// TIA Portal project "磬苑一队（6部十层）" (V15.1)

(* hardware
DEVICE "S7-1200 station_1"  S7-1200 Station
   slot 0: "Rack_0"  S7-1200 Rack  Rack  V1.0
   slot 1: "PLC_1"  CPU 1215C DC/DC/DC  6ES7 215-1AG40-0XB0  V4.2
DEVICE "PC-System_1"  SIMATIC PC station
   slot 0: "SIMATIC PC station"  Rail  SIMATIC PC-Station  V1.0
      slot 125: "Stationmanager"  Station_Manager  V6.0.4
   slot 1: "IE general_1"  IE General  IE_CP  V8.2.0
*)

// ===== PLC "PLC_1"  CPU 1215C DC/DC/DC =====

VAR_GLOBAL   // PLC tag table "默认变量表"
   "输入自动运行信号" AT %M0.0 : Bool;
   "Tag_1" AT %M100.0 : Bool;
   "Clock_Byte" AT %MB0 : Byte;
   "Clock_5Hz" AT %M0.1 : Bool;
   "Clock_2.5Hz" AT %M0.2 : Bool;
   "Clock_2Hz" AT %M0.3 : Bool;
   "Clock_1.25Hz" AT %M0.4 : Bool;
   "Clock_1Hz" AT %M0.5 : Bool;
   "Clock_0.625Hz" AT %M0.6 : Bool;
   "Clock_0.5Hz" AT %M0.7 : Bool;
END_VAR

DATA_BLOCK "IN"   // DB1
{ S7_Optimized_Access := 'FALSE' }
VERSION : 0.1
   VAR
      "1层上行呼梯按钮" : Bool := FALSE;
      "2层上行呼梯按钮" : Bool := FALSE;
      "3层上行呼梯按钮" : Bool := FALSE;
      "4层上行呼梯按钮" : Bool := FALSE;
      "5层上行呼梯按钮" : Bool := FALSE;
      "6层上行呼梯按钮" : Bool := FALSE;
      "7层上行呼梯按钮" : Bool := FALSE;
      "8层上行呼梯按钮" : Bool := FALSE;
      "9层上行呼梯按钮" : Bool := FALSE;
      "2层下行呼梯按钮" : Bool := FALSE;
      "3层下行呼梯按钮" : Bool := FALSE;
      "4层下行呼梯按钮" : Bool := FALSE;
      "5层下行呼梯按钮" : Bool := FALSE;
      "6层下行呼梯按钮" : Bool := FALSE;
      "7层下行呼梯按钮" : Bool := FALSE;
      "8层下行呼梯按钮" : Bool := FALSE;
      "9层下行呼梯按钮" : Bool := FALSE;
      "10层下行呼梯按钮" : Bool := FALSE;
      "1号梯轿内选层按钮1" : Bool := FALSE;
      "1号梯轿内选层按钮2" : Bool := FALSE;
      "1号梯轿内选层按钮3" : Bool := FALSE;
      "1号梯轿内选层按钮4" : Bool := FALSE;
      "1号梯轿内选层按钮5" : Bool := FALSE;
      "1号梯轿内选层按钮6" : Bool := FALSE;
      "1号梯轿内选层按钮7" : Bool := FALSE;
      "1号梯轿内选层按钮8" : Bool := FALSE;
      "1号梯轿内选层按钮9" : Bool := FALSE;
      "1号梯轿内选层按钮10" : Bool := FALSE;
      "1号梯轿内开门按钮" : Bool := FALSE;
      "1号梯轿内关门按钮" : Bool := FALSE;
      "1号梯光幕信号" : Bool := FALSE;
      "1号梯检修信号" : Bool := FALSE;
      "1号梯轿厢门锁信号" : Bool := FALSE;
      "1号梯1楼层门锁信号" : Bool := FALSE;
      "1号梯2楼层门锁信号" : Bool := FALSE;
      "1号梯3楼层门锁信号" : Bool := FALSE;
      "1号梯4楼层门锁信号" : Bool := FALSE;
      "1号梯5楼层门锁信号" : Bool := FALSE;
      "1号梯6楼层门锁信号" : Bool := FALSE;
      "1号梯7楼层门锁信号" : Bool := FALSE;
      "1号梯8楼层门锁信号" : Bool := FALSE;
      "1号梯9楼层门锁信号" : Bool := FALSE;
      "1号梯10楼层门锁信号" : Bool := FALSE;
      "1号梯开门到位" : Bool := FALSE;
      "1号梯关门到位" : Bool := FALSE;
      "1号梯上平层信号" : Bool := FALSE;
      "1号梯下平层信号" : Bool := FALSE;
      "1号梯上端站第1限位" : Bool := FALSE;
      "1号梯上端站第2限位" : Bool := FALSE;
      "1号梯下端站第1限位" : Bool := FALSE;
      "1号梯下端站第2限位" : Bool := FALSE;
      "2号梯轿内选层按钮1" : Bool := FALSE;
      "2号梯轿内选层按钮2" : Bool := FALSE;
      "2号梯轿内选层按钮3" : Bool := FALSE;
      "2号梯轿内选层按钮4" : Bool := FALSE;
      "2号梯轿内选层按钮5" : Bool := FALSE;
      "2号梯轿内选层按钮6" : Bool := FALSE;
      "2号梯轿内选层按钮7" : Bool := FALSE;
      "2号梯轿内选层按钮8" : Bool := FALSE;
      "2号梯轿内选层按钮9" : Bool := FALSE;
      "2号梯轿内选层按钮10" : Bool := FALSE;
      "2号梯轿内开门按钮" : Bool := FALSE;
      "2号梯轿内关门按钮" : Bool := FALSE;
      "2号梯光幕信号" : Bool := FALSE;
      "2号梯检修信号" : Bool := FALSE;
      "2号梯轿厢门锁信号" : Bool := FALSE;
      "2号梯1楼层门锁信号" : Bool := FALSE;
      "2号梯2楼层门锁信号" : Bool := FALSE;
      "2号梯3楼层门锁信号" : Bool := FALSE;
      "2号梯4楼层门锁信号" : Bool := FALSE;
      "2号梯5楼层门锁信号" : Bool := FALSE;
      "2号梯6楼层门锁信号" : Bool := FALSE;
      "2号梯7楼层门锁信号" : Bool := FALSE;
      "2号梯8楼层门锁信号" : Bool := FALSE;
      "2号梯9楼层门锁信号" : Bool := FALSE;
      "2号梯10楼层门锁信号" : Bool := FALSE;
      "2号梯开门到位" : Bool := FALSE;
      "2号梯关门到位" : Bool := FALSE;
      "2号梯上平层信号" : Bool := FALSE;
      "2号梯下平层信号" : Bool := FALSE;
      "2号梯上端站第1限位" : Bool := FALSE;
      "2号梯上端站第2限位" : Bool := FALSE;
      "2号梯下端站第1限位" : Bool := FALSE;
      "2号梯下端站第2限位" : Bool := FALSE;
      "3号梯轿内选层按钮1" : Bool := FALSE;
      "3号梯轿内选层按钮2" : Bool := FALSE;
      "3号梯轿内选层按钮3" : Bool := FALSE;
      "3号梯轿内选层按钮4" : Bool := FALSE;
      "3号梯轿内选层按钮5" : Bool := FALSE;
      "3号梯轿内选层按钮6" : Bool := FALSE;
      "3号梯轿内选层按钮7" : Bool := FALSE;
      "3号梯轿内选层按钮8" : Bool := FALSE;
      "3号梯轿内选层按钮9" : Bool := FALSE;
      "3号梯轿内选层按钮10" : Bool := FALSE;
      "3号梯轿内开门按钮" : Bool := FALSE;
      "3号梯轿内关门按钮" : Bool := FALSE;
      "3号梯光幕信号" : Bool := FALSE;
      "3号梯检修信号" : Bool := FALSE;
      "3号梯轿厢门锁信号" : Bool := FALSE;
      "3号梯1楼层门锁信号" : Bool := FALSE;
      "3号梯2楼层门锁信号" : Bool := FALSE;
      "3号梯3楼层门锁信号" : Bool := FALSE;
      "3号梯4楼层门锁信号" : Bool := FALSE;
      "3号梯5楼层门锁信号" : Bool := FALSE;
      "3号梯6楼层门锁信号" : Bool := FALSE;
      "3号梯7楼层门锁信号" : Bool := FALSE;
      "3号梯8楼层门锁信号" : Bool := FALSE;
      "3号梯9楼层门锁信号" : Bool := FALSE;
      "3号梯10楼层门锁信号" : Bool := FALSE;
      "3号梯开门到位" : Bool := FALSE;
      "3号梯关门到位" : Bool := FALSE;
      "3号梯上平层信号" : Bool := FALSE;
      "3号梯下平层信号" : Bool := FALSE;
      "3号梯上端站第1限位" : Bool := FALSE;
      "3号梯上端站第2限位" : Bool := FALSE;
      "3号梯下端站第1限位" : Bool := FALSE;
      "3号梯下端站第2限位" : Bool := FALSE;
      "4号梯轿内选层按钮1" : Bool := FALSE;
      "4号梯轿内选层按钮2" : Bool := FALSE;
      "4号梯轿内选层按钮3" : Bool := FALSE;
      "4号梯轿内选层按钮4" : Bool := FALSE;
      "4号梯轿内选层按钮5" : Bool := FALSE;
      "4号梯轿内选层按钮6" : Bool := FALSE;
      "4号梯轿内选层按钮7" : Bool := FALSE;
      "4号梯轿内选层按钮8" : Bool := FALSE;
      "4号梯轿内选层按钮9" : Bool := FALSE;
      "4号梯轿内选层按钮10" : Bool := FALSE;
      "4号梯轿内开门按钮" : Bool := FALSE;
      "4号梯轿内关门按钮" : Bool := FALSE;
      "4号梯光幕信号" : Bool := FALSE;
      "4号梯检修信号" : Bool := FALSE;
      "4号梯轿厢门锁信号" : Bool := FALSE;
      "4号梯1楼层门锁信号" : Bool := FALSE;
      "4号梯2楼层门锁信号" : Bool := FALSE;
      "4号梯3楼层门锁信号" : Bool := FALSE;
      "4号梯4楼层门锁信号" : Bool := FALSE;
      "4号梯5楼层门锁信号" : Bool := FALSE;
      "4号梯6楼层门锁信号" : Bool := FALSE;
      "4号梯7楼层门锁信号" : Bool := FALSE;
      "4号梯8楼层门锁信号" : Bool := FALSE;
      "4号梯9楼层门锁信号" : Bool := FALSE;
      "4号梯10楼层门锁信号" : Bool := FALSE;
      "4号梯开门到位" : Bool := FALSE;
      "4号梯关门到位" : Bool := FALSE;
      "4号梯上平层信号" : Bool := FALSE;
      "4号梯下平层信号" : Bool := FALSE;
      "4号梯上端站第1限位" : Bool := FALSE;
      "4号梯上端站第2限位" : Bool := FALSE;
      "4号梯下端站第1限位" : Bool := FALSE;
      "4号梯下端站第2限位" : Bool := FALSE;
      "5号梯轿内选层按钮1" : Bool := FALSE;
      "5号梯轿内选层按钮2" : Bool := FALSE;
      "5号梯轿内选层按钮3" : Bool := FALSE;
      "5号梯轿内选层按钮4" : Bool := FALSE;
      "5号梯轿内选层按钮5" : Bool := FALSE;
      "5号梯轿内选层按钮6" : Bool := FALSE;
      "5号梯轿内选层按钮7" : Bool := FALSE;
      "5号梯轿内选层按钮8" : Bool := FALSE;
      "5号梯轿内选层按钮9" : Bool := FALSE;
      "5号梯轿内选层按钮10" : Bool := FALSE;
      "5号梯轿内开门按钮" : Bool := FALSE;
      "5号梯轿内关门按钮" : Bool := FALSE;
      "5号梯光幕信号" : Bool := FALSE;
      "5号梯检修信号" : Bool := FALSE;
      "5号梯轿厢门锁信号" : Bool := FALSE;
      "5号梯1楼层门锁信号" : Bool := FALSE;
      "5号梯2楼层门锁信号" : Bool := FALSE;
      "5号梯3楼层门锁信号" : Bool := FALSE;
      "5号梯4楼层门锁信号" : Bool := FALSE;
      "5号梯5楼层门锁信号" : Bool := FALSE;
      "5号梯6楼层门锁信号" : Bool := FALSE;
      "5号梯7楼层门锁信号" : Bool := FALSE;
      "5号梯8楼层门锁信号" : Bool := FALSE;
      "5号梯9楼层门锁信号" : Bool := FALSE;
      "5号梯10楼层门锁信号" : Bool := FALSE;
      "5号梯开门到位" : Bool := FALSE;
      "5号梯关门到位" : Bool := FALSE;
      "5号梯上平层信号" : Bool := FALSE;
      "5号梯下平层信号" : Bool := FALSE;
      "5号梯上端站第1限位" : Bool := FALSE;
      "5号梯上端站第2限位" : Bool := FALSE;
      "5号梯下端站第1限位" : Bool := FALSE;
      "5号梯下端站第2限位" : Bool := FALSE;
      "6号梯轿内选层按钮1" : Bool := FALSE;
      "6号梯轿内选层按钮2" : Bool := FALSE;
      "6号梯轿内选层按钮3" : Bool := FALSE;
      "6号梯轿内选层按钮4" : Bool := FALSE;
      "6号梯轿内选层按钮5" : Bool := FALSE;
      "6号梯轿内选层按钮6" : Bool := FALSE;
      "6号梯轿内选层按钮7" : Bool := FALSE;
      "6号梯轿内选层按钮8" : Bool := FALSE;
      "6号梯轿内选层按钮9" : Bool := FALSE;
      "6号梯轿内选层按钮10" : Bool := FALSE;
      "6号梯轿内开门按钮" : Bool := FALSE;
      "6号梯轿内关门按钮" : Bool := FALSE;
      "6号梯光幕信号" : Bool := FALSE;
      "6号梯检修信号" : Bool := FALSE;
      "6号梯轿厢门锁信号" : Bool := FALSE;
      "6号梯1楼层门锁信号" : Bool := FALSE;
      "6号梯2楼层门锁信号" : Bool := FALSE;
      "6号梯3楼层门锁信号" : Bool := FALSE;
      "6号梯4楼层门锁信号" : Bool := FALSE;
      "6号梯5楼层门锁信号" : Bool := FALSE;
      "6号梯6楼层门锁信号" : Bool := FALSE;
      "6号梯7楼层门锁信号" : Bool := FALSE;
      "6号梯8楼层门锁信号" : Bool := FALSE;
      "6号梯9楼层门锁信号" : Bool := FALSE;
      "6号梯10楼层门锁信号" : Bool := FALSE;
      "6号梯开门到位" : Bool := FALSE;
      "6号梯关门到位" : Bool := FALSE;
      "6号梯上平层信号" : Bool := FALSE;
      "6号梯下平层信号" : Bool := FALSE;
      "6号梯上端站第1限位" : Bool := FALSE;
      "6号梯上端站第2限位" : Bool := FALSE;
      "6号梯下端站第1限位" : Bool := FALSE;
      "6号梯下端站第2限位" : Bool := FALSE;
      自动运行信号 : Bool := FALSE;
      "1号梯当前载重量" : Word := 0;
      "2号梯当前载重量" : Word := 0;
      "3号梯当前载重量" : Word := 0;
      "4号梯当前载重量" : Word := 0;
      "5号梯当前载重量" : Word := 0;
      "6号梯当前载重量" : Word := 0;
   END_VAR
BEGIN
END_DATA_BLOCK

DATA_BLOCK "OUT"   // DB2
{ S7_Optimized_Access := 'FALSE' }
VERSION : 0.1
   VAR
      "1层上行呼梯按钮指示灯" : Bool := FALSE;
      "2层上行呼梯按钮指示灯" : Bool := FALSE;
      "3层上行呼梯按钮指示灯" : Bool := FALSE;
      "4层上行呼梯按钮指示灯" : Bool := FALSE;
      "5层上行呼梯按钮指示灯" : Bool := FALSE;
      "6层上行呼梯按钮指示灯" : Bool := FALSE;
      "7层上行呼梯按钮指示灯" : Bool := FALSE;
      "8层上行呼梯按钮指示灯" : Bool := FALSE;
      "9层上行呼梯按钮指示灯" : Bool := FALSE;
      "2层下行呼梯按钮指示灯" : Bool := FALSE;
      "3层下行呼梯按钮指示灯" : Bool := FALSE;
      "4层下行呼梯按钮指示灯" : Bool := FALSE;
      "5层下行呼梯按钮指示灯" : Bool := FALSE;
      "6层下行呼梯按钮指示灯" : Bool := FALSE;
      "7层下行呼梯按钮指示灯" : Bool := FALSE;
      "8层下行呼梯按钮指示灯" : Bool := FALSE;
      "9层下行呼梯按钮指示灯" : Bool := FALSE;
      "10层下行呼梯按钮指示灯" : Bool := FALSE;
      "1号梯1层按钮指示灯" : Bool := FALSE;
      "1号梯2层按钮指示灯" : Bool := FALSE;
      "1号梯3层按钮指示灯" : Bool := FALSE;
      "1号梯4层按钮指示灯" : Bool := FALSE;
      "1号梯5层按钮指示灯" : Bool := FALSE;
      "1号梯6层按钮指示灯" : Bool := FALSE;
      "1号梯7层按钮指示灯" : Bool := FALSE;
      "1号梯8层按钮指示灯" : Bool := FALSE;
      "1号梯9层按钮指示灯" : Bool := FALSE;
      "1号梯10层按钮指示灯" : Bool := FALSE;
      "1号梯LEDa" : Bool := FALSE;
      "1号梯LEDb" : Bool := FALSE;
      "1号梯LEDc" : Bool := FALSE;
      "1号梯LEDd" : Bool := FALSE;
      "1号梯LEDe" : Bool := FALSE;
      "1号梯LEDf" : Bool := FALSE;
      "1号梯LEDg" : Bool := FALSE;
      "1号梯LEDh" : Bool := FALSE;
      "1号梯LEDi" : Bool := FALSE;
      "1号梯LEDj" : Bool := FALSE;
      "1号梯LEDk" : Bool := FALSE;
      "1号梯LEDl" : Bool := FALSE;
      "1号梯LEDm" : Bool := FALSE;
      "1号梯LEDn" : Bool := FALSE;
      "1号梯上行指示" : Bool := FALSE;
      "1号梯下行指示" : Bool := FALSE;
      "1号梯故障指示" : Bool := FALSE;
      "1号梯照明指示" : Bool := FALSE;
      "1号梯风扇指示" : Bool := FALSE;
      "1号梯满载指示" : Bool := FALSE;
      "1号梯电机启动信号" : Bool := FALSE;
      "1号梯上行接触器" : Bool := FALSE;
      "1号梯下行接触器" : Bool := FALSE;
      "1号梯高速接触器" : Bool := FALSE;
      "1号梯低速接触器" : Bool := FALSE;
      "1号梯开门继电器" : Bool := FALSE;
      "1号梯关门继电器" : Bool := FALSE;
      "1号梯1级减速制动" : Bool := FALSE;
      "1号梯2级减速制动" : Bool := FALSE;
      "1号梯3级减速制动" : Bool := FALSE;
      "2号梯1层按钮指示灯" : Bool := FALSE;
      "2号梯2层按钮指示灯" : Bool := FALSE;
      "2号梯3层按钮指示灯" : Bool := FALSE;
      "2号梯4层按钮指示灯" : Bool := FALSE;
      "2号梯5层按钮指示灯" : Bool := FALSE;
      "2号梯6层按钮指示灯" : Bool := FALSE;
      "2号梯7层按钮指示灯" : Bool := FALSE;
      "2号梯8层按钮指示灯" : Bool := FALSE;
      "2号梯9层按钮指示灯" : Bool := FALSE;
      "2号梯10层按钮指示灯" : Bool := FALSE;
      "2号梯LEDa" : Bool := FALSE;
      "2号梯LEDb" : Bool := FALSE;
      "2号梯LEDc" : Bool := FALSE;
      "2号梯LEDd" : Bool := FALSE;
      "2号梯LEDe" : Bool := FALSE;
      "2号梯LEDf" : Bool := FALSE;
      "2号梯LEDg" : Bool := FALSE;
      "2号梯LEDh" : Bool := FALSE;
      "2号梯LEDi" : Bool := FALSE;
      "2号梯LEDj" : Bool := FALSE;
      "2号梯LEDk" : Bool := FALSE;
      "2号梯LEDl" : Bool := FALSE;
      "2号梯LEDm" : Bool := FALSE;
      "2号梯LEDn" : Bool := FALSE;
      "2号梯上行指示" : Bool := FALSE;
      "2号梯下行指示" : Bool := FALSE;
      "2号梯故障指示" : Bool := FALSE;
      "2号梯照明指示" : Bool := FALSE;
      "2号梯风扇指示" : Bool := FALSE;
      "2号梯满载指示" : Bool := FALSE;
      "2号梯电机启动信号" : Bool := FALSE;
      "2号梯上行接触器" : Bool := FALSE;
      "2号梯下行接触器" : Bool := FALSE;
      "2号梯高速接触器" : Bool := FALSE;
      "2号梯低速接触器" : Bool := FALSE;
      "2号梯开门继电器" : Bool := FALSE;
      "2号梯关门继电器" : Bool := FALSE;
      "2号梯1级减速制动" : Bool := FALSE;
      "2号梯2级减速制动" : Bool := FALSE;
      "2号梯3级减速制动" : Bool := FALSE;
      "3号梯1层按钮指示灯" : Bool := FALSE;
      "3号梯2层按钮指示灯" : Bool := FALSE;
      "3号梯3层按钮指示灯" : Bool := FALSE;
      "3号梯4层按钮指示灯" : Bool := FALSE;
      "3号梯5层按钮指示灯" : Bool := FALSE;
      "3号梯6层按钮指示灯" : Bool := FALSE;
      "3号梯7层按钮指示灯" : Bool := FALSE;
      "3号梯8层按钮指示灯" : Bool := FALSE;
      "3号梯9层按钮指示灯" : Bool := FALSE;
      "3号梯10层按钮指示灯" : Bool := FALSE;
      "3号梯LEDa" : Bool := FALSE;
      "3号梯LEDb" : Bool := FALSE;
      "3号梯LEDc" : Bool := FALSE;
      "3号梯LEDd" : Bool := FALSE;
      "3号梯LEDe" : Bool := FALSE;
      "3号梯LEDf" : Bool := FALSE;
      "3号梯LEDg" : Bool := FALSE;
      "3号梯LEDh" : Bool := FALSE;
      "3号梯LEDi" : Bool := FALSE;
      "3号梯LEDj" : Bool := FALSE;
      "3号梯LEDk" : Bool := FALSE;
      "3号梯LEDl" : Bool := FALSE;
      "3号梯LEDm" : Bool := FALSE;
      "3号梯LEDn" : Bool := FALSE;
      "3号梯上行指示" : Bool := FALSE;
      "3号梯下行指示" : Bool := FALSE;
      "3号梯故障指示" : Bool := FALSE;
      "3号梯照明指示" : Bool := FALSE;
      "3号梯风扇指示" : Bool := FALSE;
      "3号梯满载指示" : Bool := FALSE;
      "3号梯电机启动信号" : Bool := FALSE;
      "3号梯上行接触器" : Bool := FALSE;
      "3号梯下行接触器" : Bool := FALSE;
      "3号梯高速接触器" : Bool := FALSE;
      "3号梯低速接触器" : Bool := FALSE;
      "3号梯开门继电器" : Bool := FALSE;
      "3号梯关门继电器" : Bool := FALSE;
      "3号梯1级减速制动" : Bool := FALSE;
      "3号梯2级减速制动" : Bool := FALSE;
      "3号梯3级减速制动" : Bool := FALSE;
      "4号梯1层按钮指示灯" : Bool := FALSE;
      "4号梯2层按钮指示灯" : Bool := FALSE;
      "4号梯3层按钮指示灯" : Bool := FALSE;
      "4号梯4层按钮指示灯" : Bool := FALSE;
      "4号梯5层按钮指示灯" : Bool := FALSE;
      "4号梯6层按钮指示灯" : Bool := FALSE;
      "4号梯7层按钮指示灯" : Bool := FALSE;
      "4号梯8层按钮指示灯" : Bool := FALSE;
      "4号梯9层按钮指示灯" : Bool := FALSE;
      "4号梯10层按钮指示灯" : Bool := FALSE;
      "4号梯LEDa" : Bool := FALSE;
      "4号梯LEDb" : Bool := FALSE;
      "4号梯LEDc" : Bool := FALSE;
      "4号梯LEDd" : Bool := FALSE;
      "4号梯LEDe" : Bool := FALSE;
      "4号梯LEDf" : Bool := FALSE;
      "4号梯LEDg" : Bool := FALSE;
      "4号梯LEDh" : Bool := FALSE;
      "4号梯LEDi" : Bool := FALSE;
      "4号梯LEDj" : Bool := FALSE;
      "4号梯LEDk" : Bool := FALSE;
      "4号梯LEDl" : Bool := FALSE;
      "4号梯LEDm" : Bool := FALSE;
      "4号梯LEDn" : Bool := FALSE;
      "4号梯上行指示" : Bool := FALSE;
      "4号梯下行指示" : Bool := FALSE;
      "4号梯故障指示" : Bool := FALSE;
      "4号梯照明指示" : Bool := FALSE;
      "4号梯风扇指示" : Bool := FALSE;
      "4号梯满载指示" : Bool := FALSE;
      "4号梯电机启动信号" : Bool := FALSE;
      "4号梯上行接触器" : Bool := FALSE;
      "4号梯下行接触器" : Bool := FALSE;
      "4号梯高速接触器" : Bool := FALSE;
      "4号梯低速接触器" : Bool := FALSE;
      "4号梯开门继电器" : Bool := FALSE;
      "4号梯关门继电器" : Bool := FALSE;
      "4号梯1级减速制动" : Bool := FALSE;
      "4号梯2级减速制动" : Bool := FALSE;
      "4号梯3级减速制动" : Bool := FALSE;
      "5号梯1层按钮指示灯" : Bool := FALSE;
      "5号梯2层按钮指示灯" : Bool := FALSE;
      "5号梯3层按钮指示灯" : Bool := FALSE;
      "5号梯4层按钮指示灯" : Bool := FALSE;
      "5号梯5层按钮指示灯" : Bool := FALSE;
      "5号梯6层按钮指示灯" : Bool := FALSE;
      "5号梯7层按钮指示灯" : Bool := FALSE;
      "5号梯8层按钮指示灯" : Bool := FALSE;
      "5号梯9层按钮指示灯" : Bool := FALSE;
      "5号梯10层按钮指示灯" : Bool := FALSE;
      "5号梯LEDa" : Bool := FALSE;
      "5号梯LEDb" : Bool := FALSE;
      "5号梯LEDc" : Bool := FALSE;
      "5号梯LEDd" : Bool := FALSE;
      "5号梯LEDe" : Bool := FALSE;
      "5号梯LEDf" : Bool := FALSE;
      "5号梯LEDg" : Bool := FALSE;
      "5号梯LEDh" : Bool := FALSE;
      "5号梯LEDi" : Bool := FALSE;
      "5号梯LEDj" : Bool := FALSE;
      "5号梯LEDk" : Bool := FALSE;
      "5号梯LEDl" : Bool := FALSE;
      "5号梯LEDm" : Bool := FALSE;
      "5号梯LEDn" : Bool := FALSE;
      "5号梯上行指示" : Bool := FALSE;
      "5号梯下行指示" : Bool := FALSE;
      "5号梯故障指示" : Bool := FALSE;
      "5号梯照明指示" : Bool := FALSE;
      "5号梯风扇指示" : Bool := FALSE;
      "5号梯满载指示" : Bool := FALSE;
      "5号梯电机启动信号" : Bool := FALSE;
      "5号梯上行接触器" : Bool := FALSE;
      "5号梯下行接触器" : Bool := FALSE;
      "5号梯高速接触器" : Bool := FALSE;
      "5号梯低速接触器" : Bool := FALSE;
      "5号梯开门继电器" : Bool := FALSE;
      "5号梯关门继电器" : Bool := FALSE;
      "5号梯1级减速制动" : Bool := FALSE;
      "5号梯2级减速制动" : Bool := FALSE;
      "5号梯3级减速制动" : Bool := FALSE;
      "6号梯1层按钮指示灯" : Bool := FALSE;
      "6号梯2层按钮指示灯" : Bool := FALSE;
      "6号梯3层按钮指示灯" : Bool := FALSE;
      "6号梯4层按钮指示灯" : Bool := FALSE;
      "6号梯5层按钮指示灯" : Bool := FALSE;
      "6号梯6层按钮指示灯" : Bool := FALSE;
      "6号梯7层按钮指示灯" : Bool := FALSE;
      "6号梯8层按钮指示灯" : Bool := FALSE;
      "6号梯9层按钮指示灯" : Bool := FALSE;
      "6号梯10层按钮指示灯" : Bool := FALSE;
      "6号梯LEDa" : Bool := FALSE;
      "6号梯LEDb" : Bool := FALSE;
      "6号梯LEDc" : Bool := FALSE;
      "6号梯LEDd" : Bool := FALSE;
      "6号梯LEDe" : Bool := FALSE;
      "6号梯LEDf" : Bool := FALSE;
      "6号梯LEDg" : Bool := FALSE;
      "6号梯LEDh" : Bool := FALSE;
      "6号梯LEDi" : Bool := FALSE;
      "6号梯LEDj" : Bool := FALSE;
      "6号梯LEDk" : Bool := FALSE;
      "6号梯LEDl" : Bool := FALSE;
      "6号梯LEDm" : Bool := FALSE;
      "6号梯LEDn" : Bool := FALSE;
      "6号梯上行指示" : Bool := FALSE;
      "6号梯下行指示" : Bool := FALSE;
      "6号梯故障指示" : Bool := FALSE;
      "6号梯照明指示" : Bool := FALSE;
      "6号梯风扇指示" : Bool := FALSE;
      "6号梯满载指示" : Bool := FALSE;
      "6号梯电机启动信号" : Bool := FALSE;
      "6号梯上行接触器" : Bool := FALSE;
      "6号梯下行接触器" : Bool := FALSE;
      "6号梯高速接触器" : Bool := FALSE;
      "6号梯低速接触器" : Bool := FALSE;
      "6号梯开门继电器" : Bool := FALSE;
      "6号梯关门继电器" : Bool := FALSE;
      "6号梯1级减速制动" : Bool := FALSE;
      "6号梯2级减速制动" : Bool := FALSE;
      "6号梯3级减速制动" : Bool := FALSE;
      准备就绪信号 : Bool := FALSE;
   END_VAR
BEGIN
END_DATA_BLOCK

DATA_BLOCK "总程序"   // DB22
{ S7_Optimized_Access := 'FALSE' }
VERSION : 0.1
   VAR
      全部初始化完成 : Bool;
   END_VAR
BEGIN
END_DATA_BLOCK

// folder: 1号梯

DATA_BLOCK "1号梯数据块"   // DB16
{ S7_Optimized_Access := 'FALSE' }
VERSION : 0.1
   VAR
      "1号梯初始化楼层" : USInt := 0;
      "1号梯当前楼层" : USInt := 0;
      "1号电梯初始化方向" : Bool;
      "1号电梯向上初始化" : Bool;
      "1号电梯向下初始化" : Bool;
      "1号梯准备就绪信号" : Bool;
      "1号梯初始化楼层中间值byte" : USInt := 0;
      "1号梯楼层计数脉冲比较值（0）" : Bool;
      "1号梯初始化楼层设置flag" : Bool;
      "1号梯初始化楼层中间值bool上" : Bool;
      "1号梯初始化楼层中间值bool下" : Bool;
      "1号梯1层flag" : Bool;
      "1号梯2层flag" : Bool;
      "1号梯3层flag" : Bool;
      "1号梯4层flag" : Bool;
      "1号梯5层flag" : Bool;
      "1号梯6层flag" : Bool;
      "1号梯7层flag" : Bool;
      "1号梯8层flag" : Bool;
      "1号梯9层flag" : Bool;
      "1号梯10层flag" : Bool;
      "1号梯双平层信号" : Bool;
      "1号梯开门信号" : Bool;
      "1号梯开门过程量" : Bool;
      "1号梯关门信号" : Bool;
      "1号梯超重信号" : Bool;
      "1号梯载重" : UInt;
      "1号梯上行p" : Bool;
      "1号梯下行p" : Bool;
      "1号梯计数楼层解码" : Word;
      "1号梯计数楼层解码*2" : Word;
      "1号梯电机上下指示启动信号" : Bool;
      "1号梯目标层" : USInt;
      "1号梯上行动作" : Bool;
      "1号梯下行动作" : Bool;
      "1号梯停层tag" : Bool;
      "1号梯停层信号" : Bool;
      "1号梯消除呼梯" : Bool;
      "1号梯制动tag" : Bool;
      "1号梯检修" : Bool;
   END_VAR
BEGIN
END_DATA_BLOCK

// folder: 2号梯

DATA_BLOCK "2号梯数据块"   // DB15
{ S7_Optimized_Access := 'FALSE' }
VERSION : 0.1
   VAR
      "2号梯初始化楼层" : Byte := 0;
      "2号梯当前楼层" : Byte := 0;
      "2号电梯初始化方向" : Bool;
      "2号电梯向上初始化" : Bool;
      "2号电梯向下初始化" : Bool;
      "2号梯准备就绪信号" : Bool;
      "2号梯初始化楼层中间值byte" : Byte := 0;
      "2号梯楼层计数脉冲比较值（0）" : Bool;
      "2号梯初始化楼层设置flag" : Bool;
      "2号梯初始化楼层中间值bool上" : Bool;
      "2号梯初始化楼层中间值bool下" : Bool;
      "2号梯1层flag" : Bool;
      "2号梯2层flag" : Bool;
      "2号梯3层flag" : Bool;
      "2号梯4层flag" : Bool;
      "2号梯5层flag" : Bool;
      "2号梯6层flag" : Bool;
      "2号梯7层flag" : Bool;
      "2号梯8层flag" : Bool;
      "2号梯9层flag" : Bool;
      "2号梯10层flag" : Bool;
      "2号梯双平层信号" : Bool;
      "2号梯开门信号" : Bool;
      "2号梯开门过程量" : Bool;
      "2号梯关门信号" : Bool;
      "2号梯超重信号" : Bool;
      "2号梯载重" : UInt;
      "2号梯上行p" : Bool;
      "2号梯下行p" : Bool;
      "2号梯计数楼层解码" : Word;
      "2号梯计数楼层解码*2" : Word;
      "2号梯电机上下指示启动信号" : Bool;
      "2号梯目标层" : USInt;
      "2号梯上行动作" : Bool;
      "2号梯下行动作" : Bool;
      "2号梯停层tag" : Bool;
      "2号梯停层信号" : Bool;
      "2号梯消除呼梯" : Bool;
      "2号梯制动tag" : Bool;
      "2号梯检修" : Bool;
   END_VAR
BEGIN
END_DATA_BLOCK

// folder: 3号梯

DATA_BLOCK "3号梯数据块"   // DB17
{ S7_Optimized_Access := 'FALSE' }
VERSION : 0.1
   VAR
      "3号梯初始化楼层" : Byte := 0;
      "3号梯当前楼层" : Byte := 0;
      "3号电梯初始化方向" : Bool;
      "3号电梯向上初始化" : Bool;
      "3号电梯向下初始化" : Bool;
      "3号梯准备就绪信号" : Bool;
      "3号梯初始化楼层中间值byte" : Byte := 0;
      "3号梯楼层计数脉冲比较值（0）" : Bool;
      "3号梯初始化楼层设置flag" : Bool;
      "3号梯初始化楼层中间值bool上" : Bool;
      "3号梯初始化楼层中间值bool下" : Bool;
      "3号梯1层flag" : Bool;
      "3号梯2层flag" : Bool;
      "3号梯3层flag" : Bool;
      "3号梯4层flag" : Bool;
      "3号梯5层flag" : Bool;
      "3号梯6层flag" : Bool;
      "3号梯7层flag" : Bool;
      "3号梯8层flag" : Bool;
      "3号梯9层flag" : Bool;
      "3号梯10层flag" : Bool;
      "3号梯双平层信号" : Bool;
      "3号梯开门信号" : Bool;
      "3号梯开门过程量" : Bool;
      "3号梯关门信号" : Bool;
      "3号梯超重信号" : Bool;
      "3号梯载重" : UInt;
      "3号梯上行p" : Bool;
      "3号梯下行p" : Bool;
      "3号梯计数楼层解码" : Word;
      "3号梯计数楼层解码*2" : Word;
      "3号梯电机上下指示启动信号" : Bool;
      "3号梯目标层" : USInt;
      "3号梯上行动作" : Bool;
      "3号梯下行动作" : Bool;
      "3号梯停层tag" : Bool;
      "3号梯停层信号" : Bool;
      "3号梯消除呼梯" : Bool;
      "3号梯制动tag" : Bool;
      "3号梯检修" : Bool;
   END_VAR
BEGIN
END_DATA_BLOCK

// folder: 4号梯

DATA_BLOCK "4号梯数据块"   // DB18
{ S7_Optimized_Access := 'FALSE' }
VERSION : 0.1
   VAR
      "4号梯初始化楼层" : Byte := 0;
      "4号梯当前楼层" : Byte := 0;
      "4号电梯初始化方向" : Bool;
      "4号电梯向上初始化" : Bool;
      "4号电梯向下初始化" : Bool;
      "4号梯准备就绪信号" : Bool;
      "4号梯初始化楼层中间值byte" : Byte := 0;
      "4号梯楼层计数脉冲比较值（0）" : Bool;
      "4号梯初始化楼层设置flag" : Bool;
      "4号梯初始化楼层中间值bool上" : Bool;
      "4号梯初始化楼层中间值bool下" : Bool;
      "4号梯1层flag" : Bool;
      "4号梯2层flag" : Bool;
      "4号梯3层flag" : Bool;
      "4号梯4层flag" : Bool;
      "4号梯5层flag" : Bool;
      "4号梯6层flag" : Bool;
      "4号梯7层flag" : Bool;
      "4号梯8层flag" : Bool;
      "4号梯9层flag" : Bool;
      "4号梯10层flag" : Bool;
      "4号梯双平层信号" : Bool;
      "4号梯开门信号" : Bool;
      "4号梯开门过程量" : Bool;
      "4号梯关门信号" : Bool;
      "4号梯超重信号" : Bool;
      "4号梯载重" : UInt;
      "4号梯上行p" : Bool;
      "4号梯下行p" : Bool;
      "4号梯计数楼层解码" : Word;
      "4号梯计数楼层解码*2" : Word;
      "4号梯电机上下指示启动信号" : Bool;
      "4号梯目标层" : USInt;
      "4号梯上行动作" : Bool;
      "4号梯下行动作" : Bool;
      "4号梯停层tag" : Bool;
      "4号梯停层信号" : Bool;
      "4号梯消除呼梯" : Bool;
      "4号梯制动tag" : Bool;
      "4号梯检修" : Bool;
   END_VAR
BEGIN
END_DATA_BLOCK

// folder: 5号梯

DATA_BLOCK "5号梯数据块"   // DB19
{ S7_Optimized_Access := 'FALSE' }
VERSION : 0.1
   VAR
      "5号梯初始化楼层" : Byte := 0;
      "5号梯当前楼层" : Byte := 0;
      "5号电梯初始化方向" : Bool;
      "5号电梯向上初始化" : Bool;
      "5号电梯向下初始化" : Bool;
      "5号梯准备就绪信号" : Bool;
      "5号梯初始化楼层中间值byte" : Byte := 0;
      "5号梯楼层计数脉冲比较值（0）" : Bool;
      "5号梯初始化楼层设置flag" : Bool;
      "5号梯初始化楼层中间值bool上" : Bool;
      "5号梯初始化楼层中间值bool下" : Bool;
      "5号梯1层flag" : Bool;
      "5号梯2层flag" : Bool;
      "5号梯3层flag" : Bool;
      "5号梯4层flag" : Bool;
      "5号梯5层flag" : Bool;
      "5号梯6层flag" : Bool;
      "5号梯7层flag" : Bool;
      "5号梯8层flag" : Bool;
      "5号梯9层flag" : Bool;
      "5号梯10层flag" : Bool;
      "5号梯双平层信号" : Bool;
      "5号梯开门信号" : Bool;
      "5号梯开门过程量" : Bool;
      "5号梯关门信号" : Bool;
      "5号梯超重信号" : Bool;
      "5号梯载重" : UInt;
      "5号梯上行p" : Bool;
      "5号梯下行p" : Bool;
      "5号梯计数楼层解码" : Word;
      "5号梯计数楼层解码*2" : Word;
      "5号梯电机上下指示启动信号" : Bool;
      "5号梯目标层" : USInt;
      "5号梯上行动作" : Bool;
      "5号梯下行动作" : Bool;
      "5号梯停层tag" : Bool;
      "5号梯停层信号" : Bool;
      "5号梯消除呼梯" : Bool;
      "5号梯制动tag" : Bool;
      "5号梯检修" : Bool;
   END_VAR
BEGIN
END_DATA_BLOCK

// folder: 6号梯

DATA_BLOCK "6号梯数据块"   // DB20
{ S7_Optimized_Access := 'FALSE' }
VERSION : 0.1
   VAR
      "6号梯初始化楼层" : Byte := 0;
      "6号梯当前楼层" : Byte := 0;
      "6号电梯初始化方向" : Bool;
      "6号电梯向上初始化" : Bool;
      "6号电梯向下初始化" : Bool;
      "6号梯准备就绪信号" : Bool;
      "6号梯初始化楼层中间值byte" : Byte := 0;
      "6号梯楼层计数脉冲比较值（0）" : Bool;
      "6号梯初始化楼层设置flag" : Bool;
      "6号梯初始化楼层中间值bool上" : Bool;
      "6号梯初始化楼层中间值bool下" : Bool;
      "6号梯1层flag" : Bool;
      "6号梯2层flag" : Bool;
      "6号梯3层flag" : Bool;
      "6号梯4层flag" : Bool;
      "6号梯5层flag" : Bool;
      "6号梯6层flag" : Bool;
      "6号梯7层flag" : Bool;
      "6号梯8层flag" : Bool;
      "6号梯9层flag" : Bool;
      "6号梯10层flag" : Bool;
      "6号梯双平层信号" : Bool;
      "6号梯开门信号" : Bool;
      "6号梯开门过程量" : Bool;
      "6号梯关门信号" : Bool;
      "6号梯超重信号" : Bool;
      "6号梯载重" : UInt;
      "6号梯上行p" : Bool;
      "6号梯下行p" : Bool;
      "6号梯计数楼层解码" : Word;
      "6号梯计数楼层解码*2" : Word;
      "6号梯电机上下指示启动信号" : Bool;
      "6号梯目标层" : USInt;
      "6号梯上行动作" : Bool;
      "6号梯下行动作" : Bool;
      "6号梯停层tag" : Bool;
      "6号梯停层信号" : Bool;
      "6号梯消除呼梯" : Bool;
      "6号梯制动tag" : Bool;
      "6号梯检修" : Bool;
   END_VAR
BEGIN
END_DATA_BLOCK

// folder: System blocks/Program resources

DATA_BLOCK "1号梯下行延时"   // DB3
{ S7_Optimized_Access := 'TRUE' }
AUTHOR : Simatic
FAMILY : IEC
NAME : IEC_TMR
VERSION : 1.0
// stored: InstanceOfName IEC_TIMER
"IEC_TIMER"
BEGIN
END_DATA_BLOCK

DATA_BLOCK "1号梯上行延时"   // DB4
{ S7_Optimized_Access := 'TRUE' }
AUTHOR : Simatic
FAMILY : IEC
NAME : IEC_TMR
VERSION : 1.0
// stored: InstanceOfName IEC_TIMER
"IEC_TIMER"
BEGIN
END_DATA_BLOCK

DATA_BLOCK "2号梯上行延时"   // DB5
{ S7_Optimized_Access := 'TRUE' }
AUTHOR : Simatic
FAMILY : IEC
NAME : IEC_TMR
VERSION : 1.0
// stored: InstanceOfName IEC_TIMER
"IEC_TIMER"
BEGIN
END_DATA_BLOCK

DATA_BLOCK "2号梯下行延时"   // DB6
{ S7_Optimized_Access := 'TRUE' }
AUTHOR : Simatic
FAMILY : IEC
NAME : IEC_TMR
VERSION : 1.0
// stored: InstanceOfName IEC_TIMER
"IEC_TIMER"
BEGIN
END_DATA_BLOCK

DATA_BLOCK "3号梯上行延时"   // DB7
{ S7_Optimized_Access := 'TRUE' }
AUTHOR : Simatic
FAMILY : IEC
NAME : IEC_TMR
VERSION : 1.0
// stored: InstanceOfName IEC_TIMER
"IEC_TIMER"
BEGIN
END_DATA_BLOCK

DATA_BLOCK "3号梯下行延时"   // DB8
{ S7_Optimized_Access := 'TRUE' }
AUTHOR : Simatic
FAMILY : IEC
NAME : IEC_TMR
VERSION : 1.0
// stored: InstanceOfName IEC_TIMER
"IEC_TIMER"
BEGIN
END_DATA_BLOCK

DATA_BLOCK "4号梯上行延时"   // DB9
{ S7_Optimized_Access := 'TRUE' }
AUTHOR : Simatic
FAMILY : IEC
NAME : IEC_TMR
VERSION : 1.0
// stored: InstanceOfName IEC_TIMER
"IEC_TIMER"
BEGIN
END_DATA_BLOCK

DATA_BLOCK "4号梯下行延时"   // DB10
{ S7_Optimized_Access := 'TRUE' }
AUTHOR : Simatic
FAMILY : IEC
NAME : IEC_TMR
VERSION : 1.0
// stored: InstanceOfName IEC_TIMER
"IEC_TIMER"
BEGIN
END_DATA_BLOCK

DATA_BLOCK "5号梯上行延时"   // DB11
{ S7_Optimized_Access := 'TRUE' }
AUTHOR : Simatic
FAMILY : IEC
NAME : IEC_TMR
VERSION : 1.0
// stored: InstanceOfName IEC_TIMER
"IEC_TIMER"
BEGIN
END_DATA_BLOCK

DATA_BLOCK "5号梯下行延时"   // DB12
{ S7_Optimized_Access := 'TRUE' }
AUTHOR : Simatic
FAMILY : IEC
NAME : IEC_TMR
VERSION : 1.0
// stored: InstanceOfName IEC_TIMER
"IEC_TIMER"
BEGIN
END_DATA_BLOCK

DATA_BLOCK "6号梯上行延时"   // DB13
{ S7_Optimized_Access := 'TRUE' }
AUTHOR : Simatic
FAMILY : IEC
NAME : IEC_TMR
VERSION : 1.0
// stored: InstanceOfName IEC_TIMER
"IEC_TIMER"
BEGIN
END_DATA_BLOCK

DATA_BLOCK "6号梯下行延时"   // DB14
{ S7_Optimized_Access := 'TRUE' }
AUTHOR : Simatic
FAMILY : IEC
NAME : IEC_TMR
VERSION : 1.0
// stored: InstanceOfName IEC_TIMER
"IEC_TIMER"
BEGIN
END_DATA_BLOCK

DATA_BLOCK "IEC_Timer_0_DB"   // DB23
{ S7_Optimized_Access := 'TRUE' }
AUTHOR : Simatic
FAMILY : IEC
NAME : IEC_TMR
VERSION : 1.0
// stored: InstanceOfName IEC_TIMER
"IEC_TIMER"
BEGIN
END_DATA_BLOCK

DATA_BLOCK "1号梯开门等待定时器"   // DB24
{ S7_Optimized_Access := 'TRUE' }
AUTHOR : Simatic
FAMILY : IEC
NAME : IEC_TMR
VERSION : 1.0
// stored: InstanceOfName IEC_TIMER
"IEC_TIMER"
BEGIN
END_DATA_BLOCK

DATA_BLOCK "1号梯开关门转换"   // DB25
{ S7_Optimized_Access := 'TRUE' }
AUTHOR : Simatic
FAMILY : IEC
NAME : IEC_TMR
VERSION : 1.0
// stored: InstanceOfName IEC_TIMER
"IEC_TIMER"
BEGIN
END_DATA_BLOCK

DATA_BLOCK "1号梯楼层加减计数器"   // DB26
{ S7_Optimized_Access := 'TRUE' }
AUTHOR : Simatic
FAMILY : IEC
NAME : USCNTR
VERSION : 1.2
// stored: InstanceOfName IEC_USCOUNTER
"IEC_USCOUNTER"
BEGIN
END_DATA_BLOCK

DATA_BLOCK "1号梯制动定时器"   // DB27
{ S7_Optimized_Access := 'TRUE' }
AUTHOR : Simatic
FAMILY : IEC
NAME : IEC_TMR
VERSION : 1.0
// stored: InstanceOfName IEC_TIMER
"IEC_TIMER"
BEGIN
END_DATA_BLOCK

// folder: 群控算法

DATA_BLOCK "群控数据块"   // DB21
{ S7_Optimized_Access := 'TRUE' }
VERSION : 0.1
BEGIN
END_DATA_BLOCK

// folder: (top level)

FUNCTION "外呼信号显示" : Void   // FC13, LAD
{ S7_Optimized_Access := 'TRUE' }
VERSION : 0.1
BEGIN

REGION Network 1: 外呼上行指示灯置位
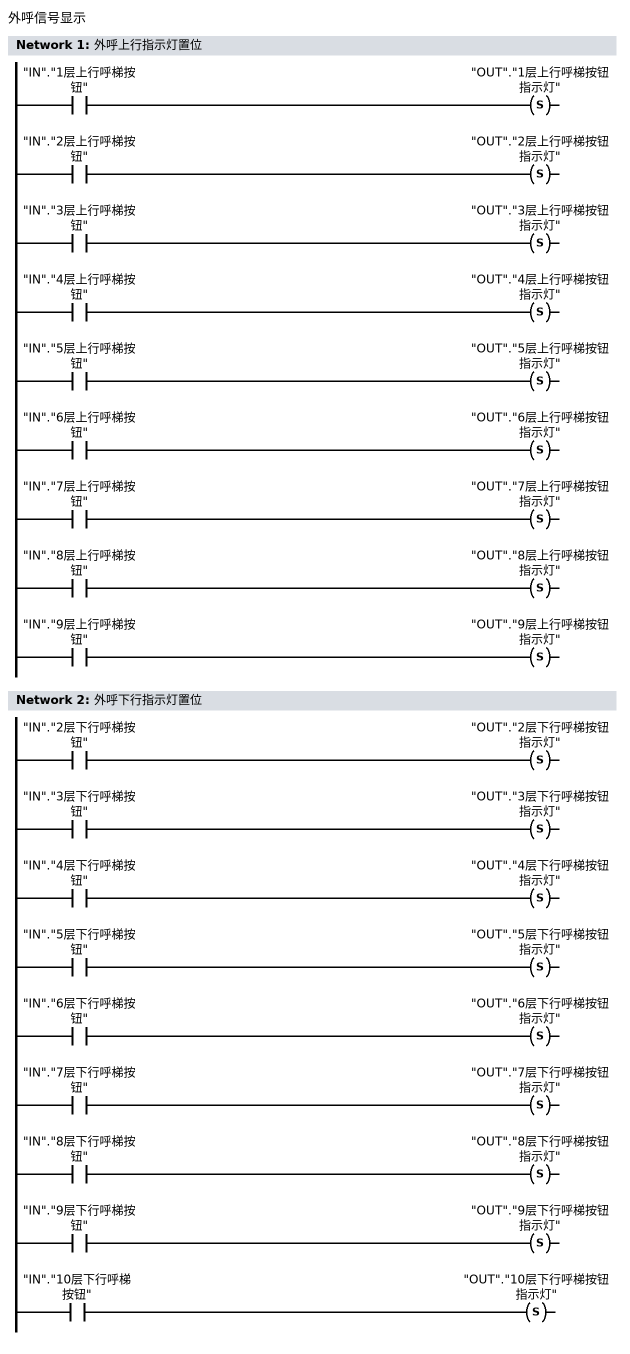
   RUNG wire#powerrail
      Contact( "IN"."1层上行呼梯按钮" )
      S_Coil( "OUT"."1层上行呼梯按钮指示灯" )
   END_RUNG
   RUNG wire#powerrail
      Contact( "IN"."2层上行呼梯按钮" )
      S_Coil( "OUT"."2层上行呼梯按钮指示灯" )
   END_RUNG
   RUNG wire#powerrail
      Contact( "IN"."3层上行呼梯按钮" )
      S_Coil( "OUT"."3层上行呼梯按钮指示灯" )
   END_RUNG
   RUNG wire#powerrail
      Contact( "IN"."4层上行呼梯按钮" )
      S_Coil( "OUT"."4层上行呼梯按钮指示灯" )
   END_RUNG
   RUNG wire#powerrail
      Contact( "IN"."5层上行呼梯按钮" )
      S_Coil( "OUT"."5层上行呼梯按钮指示灯" )
   END_RUNG
   RUNG wire#powerrail
      Contact( "IN"."6层上行呼梯按钮" )
      S_Coil( "OUT"."6层上行呼梯按钮指示灯" )
   END_RUNG
   RUNG wire#powerrail
      Contact( "IN"."7层上行呼梯按钮" )
      S_Coil( "OUT"."7层上行呼梯按钮指示灯" )
   END_RUNG
   RUNG wire#powerrail
      Contact( "IN"."8层上行呼梯按钮" )
      S_Coil( "OUT"."8层上行呼梯按钮指示灯" )
   END_RUNG
   RUNG wire#powerrail
      Contact( "IN"."9层上行呼梯按钮" )
      S_Coil( "OUT"."9层上行呼梯按钮指示灯" )
   END_RUNG
   // the same network as SCL:
   IF "IN"."1层上行呼梯按钮" THEN "OUT"."1层上行呼梯按钮指示灯" := TRUE; END_IF;
   IF "IN"."2层上行呼梯按钮" THEN "OUT"."2层上行呼梯按钮指示灯" := TRUE; END_IF;
   IF "IN"."3层上行呼梯按钮" THEN "OUT"."3层上行呼梯按钮指示灯" := TRUE; END_IF;
   IF "IN"."4层上行呼梯按钮" THEN "OUT"."4层上行呼梯按钮指示灯" := TRUE; END_IF;
   IF "IN"."5层上行呼梯按钮" THEN "OUT"."5层上行呼梯按钮指示灯" := TRUE; END_IF;
   IF "IN"."6层上行呼梯按钮" THEN "OUT"."6层上行呼梯按钮指示灯" := TRUE; END_IF;
   IF "IN"."7层上行呼梯按钮" THEN "OUT"."7层上行呼梯按钮指示灯" := TRUE; END_IF;
   IF "IN"."8层上行呼梯按钮" THEN "OUT"."8层上行呼梯按钮指示灯" := TRUE; END_IF;
   IF "IN"."9层上行呼梯按钮" THEN "OUT"."9层上行呼梯按钮指示灯" := TRUE; END_IF;
END_REGION

REGION Network 2: 外呼下行指示灯置位
   RUNG wire#powerrail
      Contact( "IN"."2层下行呼梯按钮" )
      S_Coil( "OUT"."2层下行呼梯按钮指示灯" )
   END_RUNG
   RUNG wire#powerrail
      Contact( "IN"."3层下行呼梯按钮" )
      S_Coil( "OUT"."3层下行呼梯按钮指示灯" )
   END_RUNG
   RUNG wire#powerrail
      Contact( "IN"."4层下行呼梯按钮" )
      S_Coil( "OUT"."4层下行呼梯按钮指示灯" )
   END_RUNG
   RUNG wire#powerrail
      Contact( "IN"."5层下行呼梯按钮" )
      S_Coil( "OUT"."5层下行呼梯按钮指示灯" )
   END_RUNG
   RUNG wire#powerrail
      Contact( "IN"."6层下行呼梯按钮" )
      S_Coil( "OUT"."6层下行呼梯按钮指示灯" )
   END_RUNG
   RUNG wire#powerrail
      Contact( "IN"."7层下行呼梯按钮" )
      S_Coil( "OUT"."7层下行呼梯按钮指示灯" )
   END_RUNG
   RUNG wire#powerrail
      Contact( "IN"."8层下行呼梯按钮" )
      S_Coil( "OUT"."8层下行呼梯按钮指示灯" )
   END_RUNG
   RUNG wire#powerrail
      Contact( "IN"."9层下行呼梯按钮" )
      S_Coil( "OUT"."9层下行呼梯按钮指示灯" )
   END_RUNG
   RUNG wire#powerrail
      Contact( "IN"."10层下行呼梯按钮" )
      S_Coil( "OUT"."10层下行呼梯按钮指示灯" )
   END_RUNG
   // the same network as SCL:
   IF "IN"."2层下行呼梯按钮" THEN "OUT"."2层下行呼梯按钮指示灯" := TRUE; END_IF;
   IF "IN"."3层下行呼梯按钮" THEN "OUT"."3层下行呼梯按钮指示灯" := TRUE; END_IF;
   IF "IN"."4层下行呼梯按钮" THEN "OUT"."4层下行呼梯按钮指示灯" := TRUE; END_IF;
   IF "IN"."5层下行呼梯按钮" THEN "OUT"."5层下行呼梯按钮指示灯" := TRUE; END_IF;
   IF "IN"."6层下行呼梯按钮" THEN "OUT"."6层下行呼梯按钮指示灯" := TRUE; END_IF;
   IF "IN"."7层下行呼梯按钮" THEN "OUT"."7层下行呼梯按钮指示灯" := TRUE; END_IF;
   IF "IN"."8层下行呼梯按钮" THEN "OUT"."8层下行呼梯按钮指示灯" := TRUE; END_IF;
   IF "IN"."9层下行呼梯按钮" THEN "OUT"."9层下行呼梯按钮指示灯" := TRUE; END_IF;
   IF "IN"."10层下行呼梯按钮" THEN "OUT"."10层下行呼梯按钮指示灯" := TRUE; END_IF;
END_REGION

REGION Network 3: 外呼上行指示灯复位
END_REGION

REGION Network 4: 外呼下行指示灯复位
END_REGION
END_FUNCTION

ORGANIZATION_BLOCK "Main"   // OB1, LAD, ProgramCycle
TITLE = "Main Program Sweep (Cycle)"
{ S7_Optimized_Access := 'TRUE' }
VERSION : 0.1
   VAR_INPUT
      Initial_Call : Bool;   // Initial call of this OB
      Remanence : Bool;   // =True, if remanent data are available
   END_VAR
   VAR_TEMP   // added for the SCL form of the ladder/FBD networks
      _w1 : Bool;
      _w2 : Bool;
   END_VAR
BEGIN

REGION Network 1
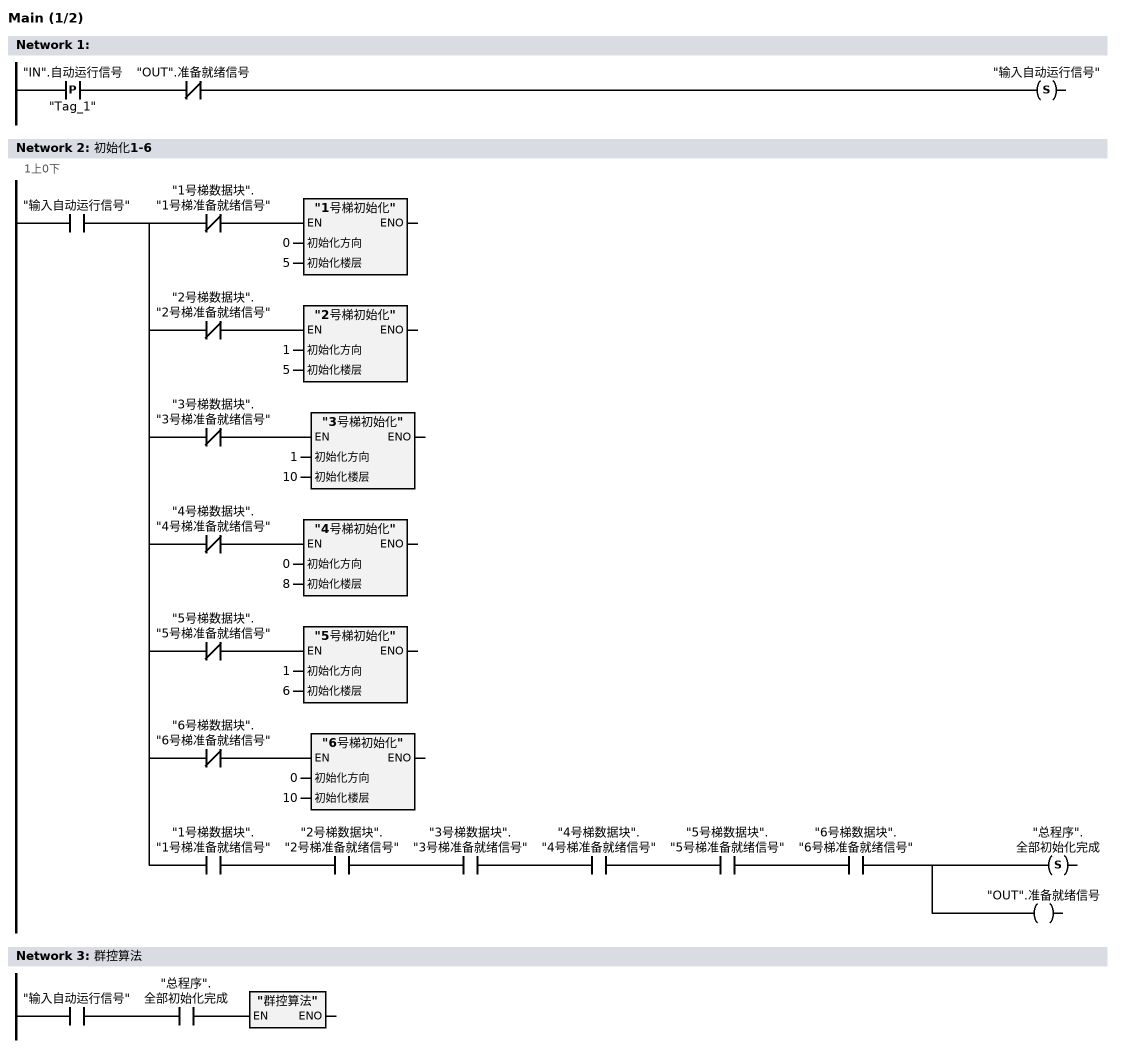
   RUNG wire#powerrail
      P_Contact(operand := "IN".自动运行信号, bit := "Tag_1")
      I_Contact( "OUT".准备就绪信号 )
      S_Coil( "输入自动运行信号" )
   END_RUNG
   // the same network as SCL:
   #_w1 := "IN".自动运行信号 AND NOT "Tag_1";   // rising edge of "IN".自动运行信号
   "Tag_1" := "IN".自动运行信号;
   IF #_w1 AND NOT "OUT".准备就绪信号 THEN "输入自动运行信号" := TRUE; END_IF;
END_REGION

REGION Network 2: 初始化1-6
   // 1上0下
   RUNG wire#powerrail
      Contact( "输入自动运行信号" )
      wire#w1
      I_Contact( "1号梯数据块"."1号梯准备就绪信号" )
      "1号梯初始化"(初始化方向 := 0, 初始化楼层 := 5)
   END_RUNG
   RUNG wire#w1
      I_Contact( "2号梯数据块"."2号梯准备就绪信号" )
      "2号梯初始化"(初始化方向 := 1, 初始化楼层 := 5)
   END_RUNG
   RUNG wire#w1
      I_Contact( "3号梯数据块"."3号梯准备就绪信号" )
      "3号梯初始化"(初始化方向 := 1, 初始化楼层 := 10)
   END_RUNG
   RUNG wire#w1
      I_Contact( "4号梯数据块"."4号梯准备就绪信号" )
      "4号梯初始化"(初始化方向 := 0, 初始化楼层 := 8)
   END_RUNG
   RUNG wire#w1
      I_Contact( "5号梯数据块"."5号梯准备就绪信号" )
      "5号梯初始化"(初始化方向 := 1, 初始化楼层 := 6)
   END_RUNG
   RUNG wire#w1
      I_Contact( "6号梯数据块"."6号梯准备就绪信号" )
      "6号梯初始化"(初始化方向 := 0, 初始化楼层 := 10)
   END_RUNG
   RUNG wire#w1
      Contact( "1号梯数据块"."1号梯准备就绪信号" )
      Contact( "2号梯数据块"."2号梯准备就绪信号" )
      Contact( "3号梯数据块"."3号梯准备就绪信号" )
      Contact( "4号梯数据块"."4号梯准备就绪信号" )
      Contact( "5号梯数据块"."5号梯准备就绪信号" )
      Contact( "6号梯数据块"."6号梯准备就绪信号" )
      wire#w2
      S_Coil( "总程序".全部初始化完成 )
   END_RUNG
   RUNG wire#w2
      Coil( "OUT".准备就绪信号 )
   END_RUNG
   // the same network as SCL:
   #_w1 := "输入自动运行信号";
   IF "输入自动运行信号" AND NOT "1号梯数据块"."1号梯准备就绪信号" THEN "1号梯初始化"(初始化方向 := 0, 初始化楼层 := 5); END_IF;
   IF #_w1 AND NOT "2号梯数据块"."2号梯准备就绪信号" THEN "2号梯初始化"(初始化方向 := 1, 初始化楼层 := 5); END_IF;
   IF #_w1 AND NOT "3号梯数据块"."3号梯准备就绪信号" THEN "3号梯初始化"(初始化方向 := 1, 初始化楼层 := 10); END_IF;
   IF #_w1 AND NOT "4号梯数据块"."4号梯准备就绪信号" THEN "4号梯初始化"(初始化方向 := 0, 初始化楼层 := 8); END_IF;
   IF #_w1 AND NOT "5号梯数据块"."5号梯准备就绪信号" THEN "5号梯初始化"(初始化方向 := 1, 初始化楼层 := 6); END_IF;
   IF #_w1 AND NOT "6号梯数据块"."6号梯准备就绪信号" THEN "6号梯初始化"(初始化方向 := 0, 初始化楼层 := 10); END_IF;
   #_w2 := #_w1 AND "1号梯数据块"."1号梯准备就绪信号" AND "2号梯数据块"."2号梯准备就绪信号" AND "3号梯数据块"."3号梯准备就绪信号" AND "4号梯数据块"."4号梯准备就绪信号" AND "5号梯数据块"."5号梯准备就绪信号" AND "6号梯数据块"."6号梯准备就绪信号";
   IF #_w2 THEN "总程序".全部初始化完成 := TRUE; END_IF;
   "OUT".准备就绪信号 := #_w2;
END_REGION

REGION Network 3: 群控算法
   RUNG wire#powerrail
      Contact( "输入自动运行信号" )
      Contact( "总程序".全部初始化完成 )
      "群控算法"()
   END_RUNG
   // the same network as SCL:
   IF "输入自动运行信号" AND "总程序".全部初始化完成 THEN "群控算法"(); END_IF;
END_REGION

REGION Network 4: 1-6显示
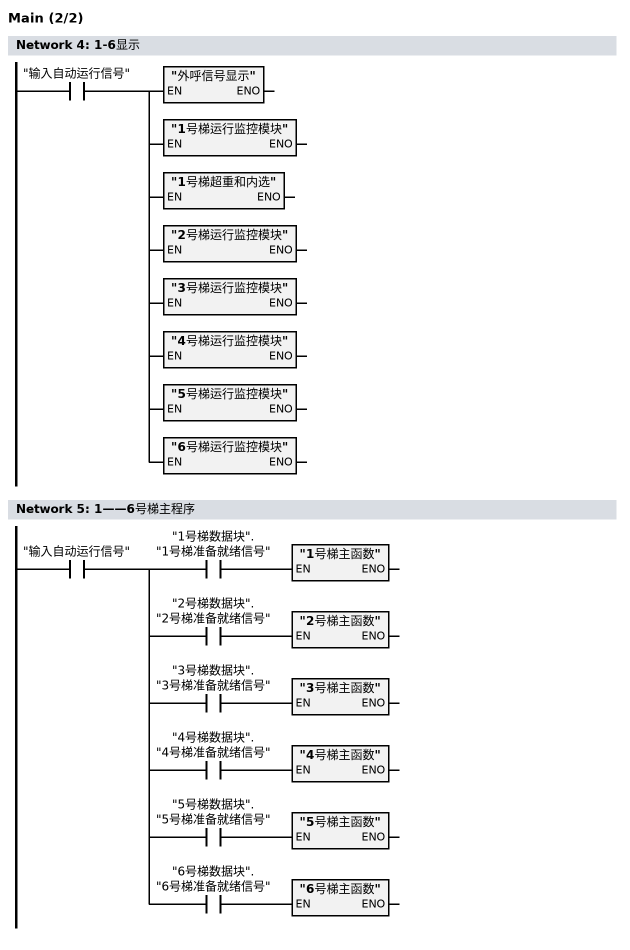
   RUNG wire#powerrail
      Contact( "输入自动运行信号" )
      wire#w1
      "外呼信号显示"()
   END_RUNG
   RUNG wire#w1
      "1号梯运行监控模块"()
   END_RUNG
   RUNG wire#w1
      "1号梯超重和内选"()
   END_RUNG
   RUNG wire#w1
      "2号梯运行监控模块"()
   END_RUNG
   RUNG wire#w1
      "3号梯运行监控模块"()
   END_RUNG
   RUNG wire#w1
      "4号梯运行监控模块"()
   END_RUNG
   RUNG wire#w1
      "5号梯运行监控模块"()
   END_RUNG
   RUNG wire#w1
      "6号梯运行监控模块"()
   END_RUNG
   RUNG wire#w1
   END_RUNG
   RUNG wire#w1
   END_RUNG
   RUNG wire#w1
   END_RUNG
   RUNG wire#w1
   END_RUNG
   RUNG wire#w1
   END_RUNG
   RUNG wire#w1
   END_RUNG
   // the same network as SCL:
   #_w1 := "输入自动运行信号";
   IF #_w1 THEN
       "外呼信号显示"();
       "1号梯运行监控模块"();
       "1号梯超重和内选"();
       "2号梯运行监控模块"();
       "3号梯运行监控模块"();
       "4号梯运行监控模块"();
       "5号梯运行监控模块"();
       "6号梯运行监控模块"();
   END_IF;
END_REGION

REGION Network 5: 1——6号梯主程序
   RUNG wire#powerrail
      Contact( "输入自动运行信号" )
      wire#w1
      Contact( "1号梯数据块"."1号梯准备就绪信号" )
      "1号梯主函数"()
   END_RUNG
   RUNG wire#w1
      Contact( "2号梯数据块"."2号梯准备就绪信号" )
      "2号梯主函数"()
   END_RUNG
   RUNG wire#w1
      Contact( "3号梯数据块"."3号梯准备就绪信号" )
      "3号梯主函数"()
   END_RUNG
   RUNG wire#w1
      Contact( "4号梯数据块"."4号梯准备就绪信号" )
      "4号梯主函数"()
   END_RUNG
   RUNG wire#w1
      Contact( "5号梯数据块"."5号梯准备就绪信号" )
      "5号梯主函数"()
   END_RUNG
   RUNG wire#w1
      Contact( "6号梯数据块"."6号梯准备就绪信号" )
      "6号梯主函数"()
   END_RUNG
   // the same network as SCL:
   #_w1 := "输入自动运行信号";
   IF "输入自动运行信号" AND "1号梯数据块"."1号梯准备就绪信号" THEN "1号梯主函数"(); END_IF;
   IF #_w1 AND "2号梯数据块"."2号梯准备就绪信号" THEN "2号梯主函数"(); END_IF;
   IF #_w1 AND "3号梯数据块"."3号梯准备就绪信号" THEN "3号梯主函数"(); END_IF;
   IF #_w1 AND "4号梯数据块"."4号梯准备就绪信号" THEN "4号梯主函数"(); END_IF;
   IF #_w1 AND "5号梯数据块"."5号梯准备就绪信号" THEN "5号梯主函数"(); END_IF;
   IF #_w1 AND "6号梯数据块"."6号梯准备就绪信号" THEN "6号梯主函数"(); END_IF;
END_REGION
END_ORGANIZATION_BLOCK

// folder: 1号梯

FUNCTION "1号梯初始化" : Void   // FC1, LAD
{ S7_Optimized_Access := 'TRUE' }
VERSION : 0.1
   VAR_INPUT
      初始化方向 : Bool;
      初始化楼层 : Byte;
   END_VAR
   VAR_TEMP   // added for the SCL form of the ladder/FBD networks
      _w1 : Bool;
      _w2 : Bool;
      _w3 : Bool;
      _w4 : Bool;
   END_VAR
BEGIN

REGION Network 1: 1号梯传参（方向+初始化楼层）
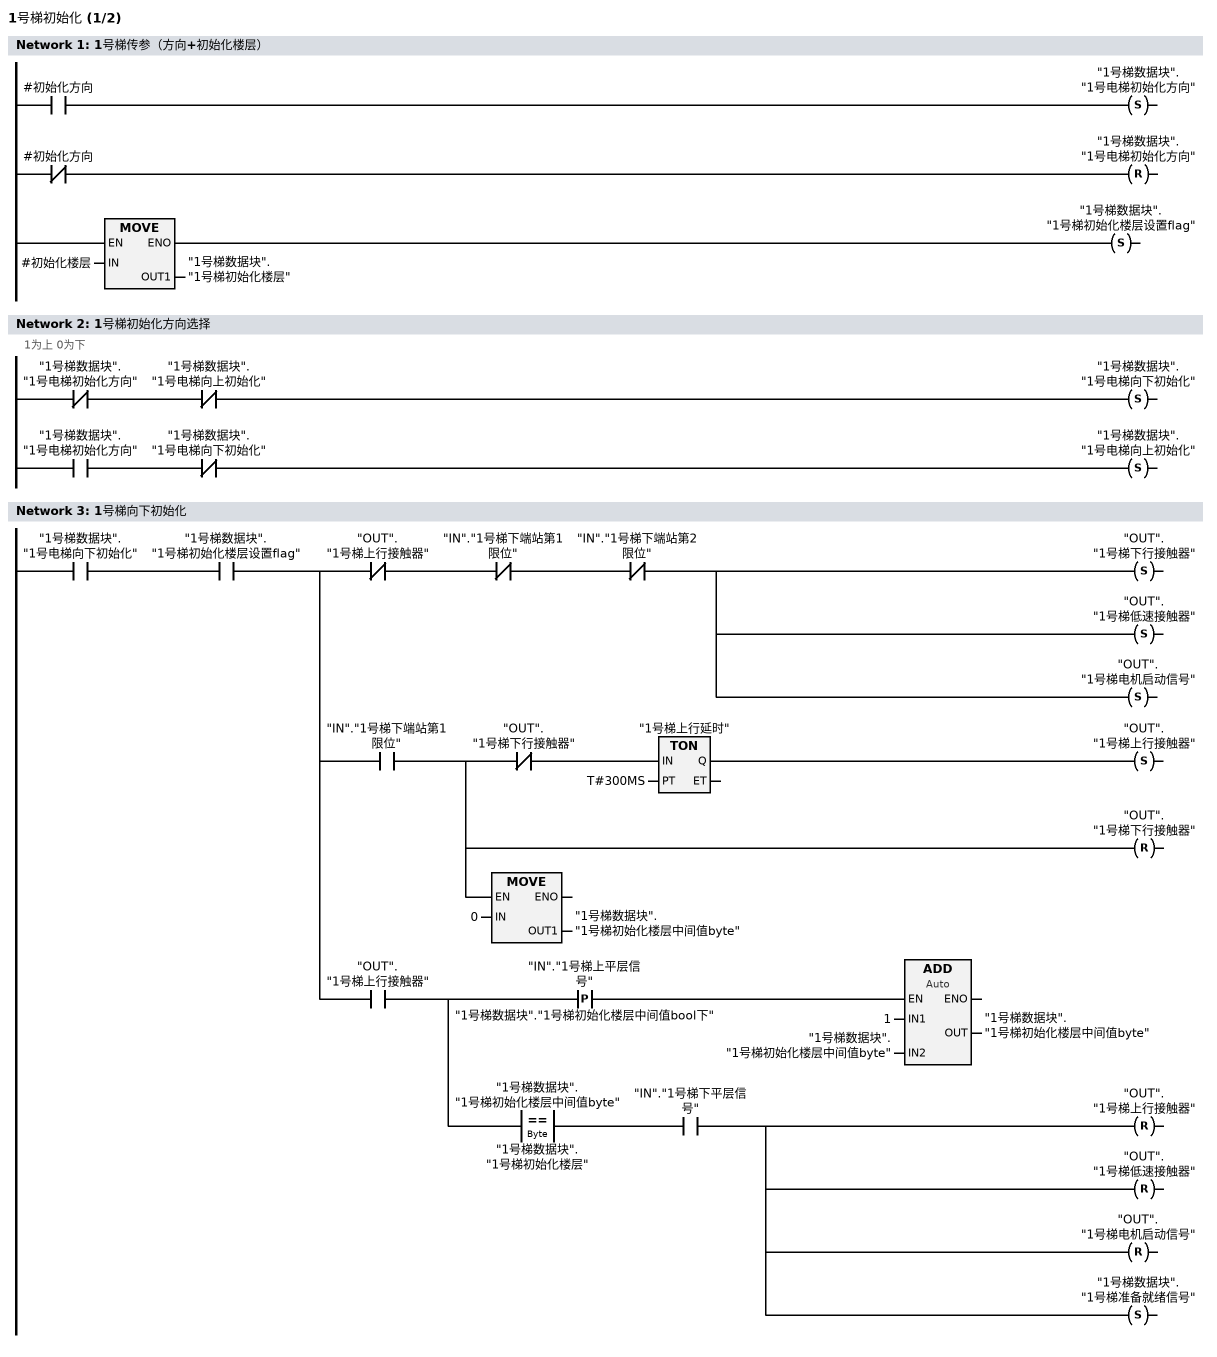
   RUNG wire#powerrail
      Contact( #初始化方向 )
      S_Coil( "1号梯数据块"."1号电梯初始化方向" )
   END_RUNG
   RUNG wire#powerrail
      I_Contact( #初始化方向 )
      R_Coil( "1号梯数据块"."1号电梯初始化方向" )
   END_RUNG
   RUNG wire#powerrail
      Move(in := #初始化楼层, out1 => "1号梯数据块"."1号梯初始化楼层")
      S_Coil( "1号梯数据块"."1号梯初始化楼层设置flag" )
   END_RUNG
   // the same network as SCL:
   IF #初始化方向 THEN "1号梯数据块"."1号电梯初始化方向" := TRUE; END_IF;
   IF NOT #初始化方向 THEN "1号梯数据块"."1号电梯初始化方向" := FALSE; END_IF;
   "1号梯数据块"."1号梯初始化楼层" := #初始化楼层;
   "1号梯数据块"."1号梯初始化楼层设置flag" := TRUE;
END_REGION

REGION Network 2: 1号梯初始化方向选择
   // 1为上 0为下
   RUNG wire#powerrail
      I_Contact( "1号梯数据块"."1号电梯初始化方向" )
      I_Contact( "1号梯数据块"."1号电梯向上初始化" )
      S_Coil( "1号梯数据块"."1号电梯向下初始化" )
   END_RUNG
   RUNG wire#powerrail
      Contact( "1号梯数据块"."1号电梯初始化方向" )
      I_Contact( "1号梯数据块"."1号电梯向下初始化" )
      S_Coil( "1号梯数据块"."1号电梯向上初始化" )
   END_RUNG
   // the same network as SCL:
   IF NOT "1号梯数据块"."1号电梯初始化方向" AND NOT "1号梯数据块"."1号电梯向上初始化" THEN "1号梯数据块"."1号电梯向下初始化" := TRUE; END_IF;
   IF "1号梯数据块"."1号电梯初始化方向" AND NOT "1号梯数据块"."1号电梯向下初始化" THEN "1号梯数据块"."1号电梯向上初始化" := TRUE; END_IF;
END_REGION

REGION Network 3: 1号梯向下初始化
   #_w1 := "1号梯数据块"."1号电梯向下初始化" AND "1号梯数据块"."1号梯初始化楼层设置flag";
   IF #_w1 AND NOT "OUT"."1号梯上行接触器" AND NOT "IN"."1号梯下端站第1限位" AND NOT "IN"."1号梯下端站第2限位" THEN
       "OUT"."1号梯下行接触器" := TRUE;
       "OUT"."1号梯低速接触器" := TRUE;
       "OUT"."1号梯电机启动信号" := TRUE;
   END_IF;
   #_w2 := #_w1 AND "IN"."1号梯下端站第1限位";
   "1号梯上行延时".TON(IN := #_w2 AND NOT "OUT"."1号梯下行接触器", PT := T#300MS);
   IF "1号梯上行延时".Q THEN "OUT"."1号梯上行接触器" := TRUE; END_IF;
   IF #_w2 THEN
       "OUT"."1号梯下行接触器" := FALSE;
       "1号梯数据块"."1号梯初始化楼层中间值byte" := 0;
   END_IF;
   #_w3 := #_w1 AND "OUT"."1号梯上行接触器";
   #_w4 := #_w3 AND "IN"."1号梯上平层信号" AND NOT "1号梯数据块"."1号梯初始化楼层中间值bool下";   // rising edge of "IN"."1号梯上平层信号"
   "1号梯数据块"."1号梯初始化楼层中间值bool下" := "IN"."1号梯上平层信号";
   IF #_w4 THEN "1号梯数据块"."1号梯初始化楼层中间值byte" := 1 + "1号梯数据块"."1号梯初始化楼层中间值byte"; END_IF;
   IF #_w3 AND ("1号梯数据块"."1号梯初始化楼层中间值byte" = "1号梯数据块"."1号梯初始化楼层") AND "IN"."1号梯下平层信号" THEN
       "OUT"."1号梯上行接触器" := FALSE;
       "OUT"."1号梯低速接触器" := FALSE;
       "OUT"."1号梯电机启动信号" := FALSE;
       "1号梯数据块"."1号梯准备就绪信号" := TRUE;
   END_IF;
END_REGION

REGION Network 4: 1号梯向上初始化
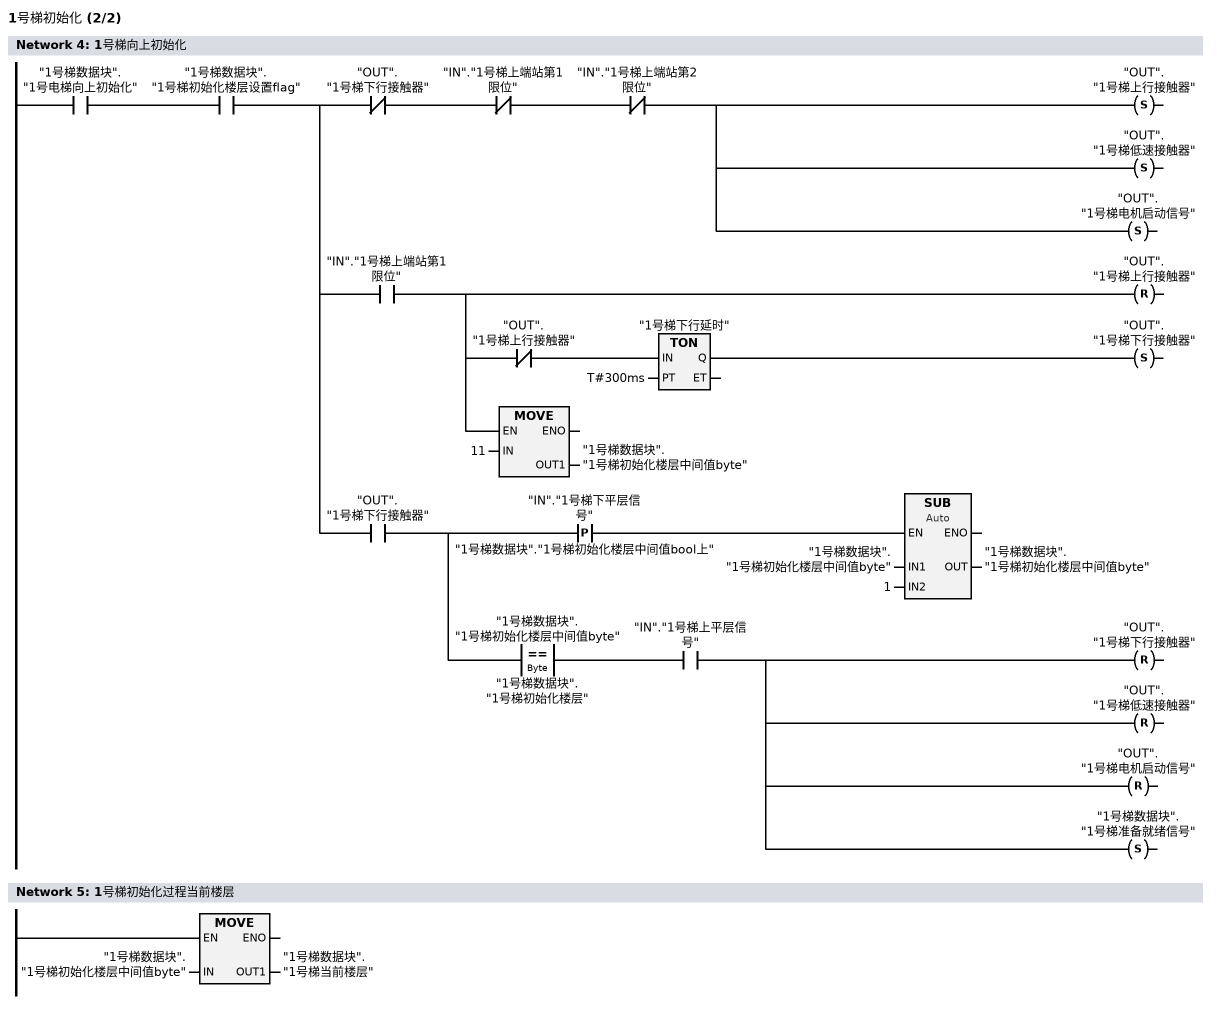
   #_w1 := "1号梯数据块"."1号电梯向上初始化" AND "1号梯数据块"."1号梯初始化楼层设置flag";
   IF #_w1 AND NOT "OUT"."1号梯下行接触器" AND NOT "IN"."1号梯上端站第1限位" AND NOT "IN"."1号梯上端站第2限位" THEN
       "OUT"."1号梯上行接触器" := TRUE;
       "OUT"."1号梯低速接触器" := TRUE;
       "OUT"."1号梯电机启动信号" := TRUE;
   END_IF;
   #_w2 := #_w1 AND "IN"."1号梯上端站第1限位";
   IF #_w2 THEN "OUT"."1号梯上行接触器" := FALSE; END_IF;
   "1号梯下行延时".TON(IN := #_w2 AND NOT "OUT"."1号梯上行接触器", PT := T#300ms);
   IF "1号梯下行延时".Q THEN "OUT"."1号梯下行接触器" := TRUE; END_IF;
   IF #_w2 THEN "1号梯数据块"."1号梯初始化楼层中间值byte" := 11; END_IF;
   #_w3 := #_w1 AND "OUT"."1号梯下行接触器";
   #_w4 := #_w3 AND "IN"."1号梯下平层信号" AND NOT "1号梯数据块"."1号梯初始化楼层中间值bool上";   // rising edge of "IN"."1号梯下平层信号"
   "1号梯数据块"."1号梯初始化楼层中间值bool上" := "IN"."1号梯下平层信号";
   IF #_w4 THEN "1号梯数据块"."1号梯初始化楼层中间值byte" := "1号梯数据块"."1号梯初始化楼层中间值byte" - 1; END_IF;
   IF #_w3 AND ("1号梯数据块"."1号梯初始化楼层中间值byte" = "1号梯数据块"."1号梯初始化楼层") AND "IN"."1号梯上平层信号" THEN
       "OUT"."1号梯下行接触器" := FALSE;
       "OUT"."1号梯低速接触器" := FALSE;
       "OUT"."1号梯电机启动信号" := FALSE;
       "1号梯数据块"."1号梯准备就绪信号" := TRUE;
   END_IF;
END_REGION

REGION Network 5: 1号梯初始化过程当前楼层
   RUNG wire#powerrail
      Move(in := "1号梯数据块"."1号梯初始化楼层中间值byte", out1 => "1号梯数据块"."1号梯当前楼层")
   END_RUNG
   // the same network as SCL:
   "1号梯数据块"."1号梯当前楼层" := "1号梯数据块"."1号梯初始化楼层中间值byte";
END_REGION
END_FUNCTION

FUNCTION "1号梯主函数" : Void   // FC8, LAD
{ S7_Optimized_Access := 'TRUE' }
VERSION : 0.1
BEGIN

REGION Network 1
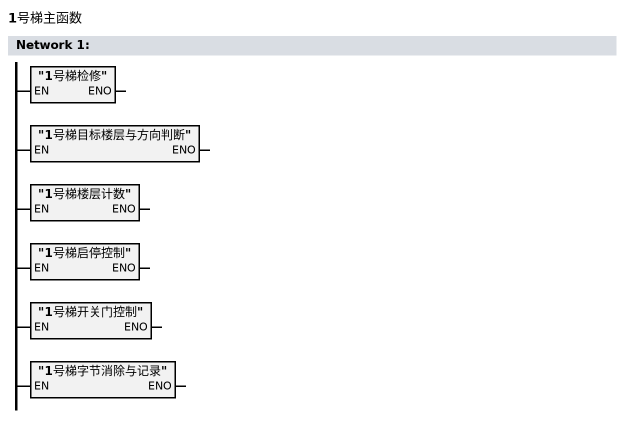
   RUNG wire#powerrail
      "1号梯检修"()
   END_RUNG
   RUNG wire#powerrail
      "1号梯目标楼层与方向判断"()
   END_RUNG
   RUNG wire#powerrail
      "1号梯楼层计数"()
   END_RUNG
   RUNG wire#powerrail
      "1号梯启停控制"()
   END_RUNG
   RUNG wire#powerrail
      "1号梯开关门控制"()
   END_RUNG
   RUNG wire#powerrail
      "1号梯字节消除与记录"()
   END_RUNG
   // the same network as SCL:
   "1号梯检修"();
   "1号梯目标楼层与方向判断"();
   "1号梯楼层计数"();
   "1号梯启停控制"();
   "1号梯开关门控制"();
   "1号梯字节消除与记录"();
END_REGION
END_FUNCTION

FUNCTION "1号梯运行监控模块" : Void   // FC14, LAD
{ S7_Optimized_Access := 'TRUE' }
VERSION : 0.1
BEGIN

REGION Network 1: 1号梯获取当前楼层设置标志位
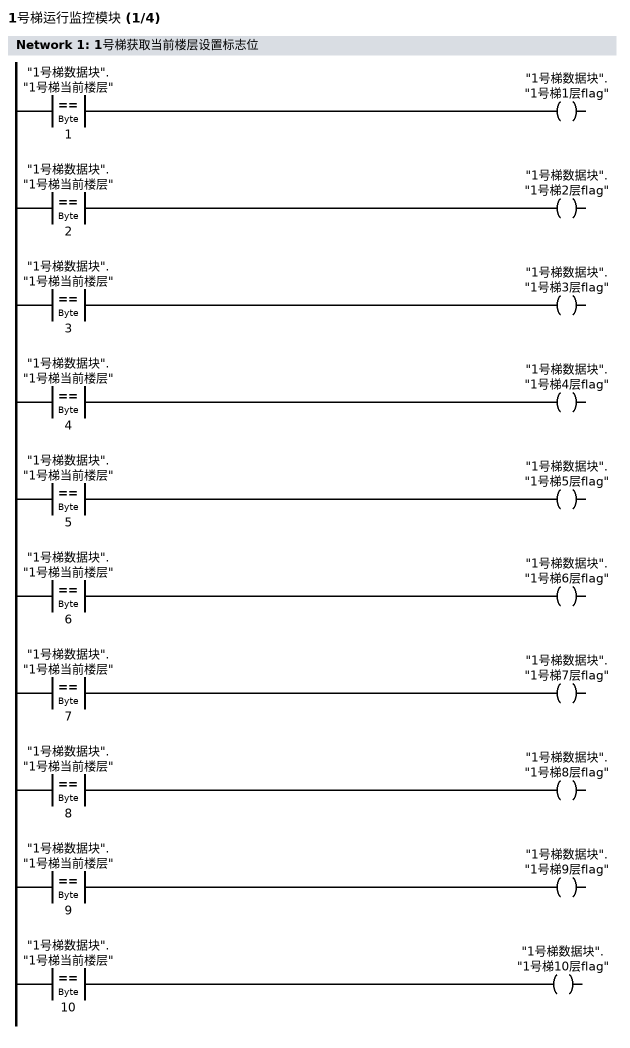
   RUNG wire#powerrail
      { S7_Templates := "SrcType := Byte" } EQ_Contact(in1 := "1号梯数据块"."1号梯当前楼层", in2 := 1)
      Coil( "1号梯数据块"."1号梯1层flag" )
   END_RUNG
   RUNG wire#powerrail
      { S7_Templates := "SrcType := Byte" } EQ_Contact(in1 := "1号梯数据块"."1号梯当前楼层", in2 := 2)
      Coil( "1号梯数据块"."1号梯2层flag" )
   END_RUNG
   RUNG wire#powerrail
      { S7_Templates := "SrcType := Byte" } EQ_Contact(in1 := "1号梯数据块"."1号梯当前楼层", in2 := 3)
      Coil( "1号梯数据块"."1号梯3层flag" )
   END_RUNG
   RUNG wire#powerrail
      { S7_Templates := "SrcType := Byte" } EQ_Contact(in1 := "1号梯数据块"."1号梯当前楼层", in2 := 4)
      Coil( "1号梯数据块"."1号梯4层flag" )
   END_RUNG
   RUNG wire#powerrail
      { S7_Templates := "SrcType := Byte" } EQ_Contact(in1 := "1号梯数据块"."1号梯当前楼层", in2 := 5)
      Coil( "1号梯数据块"."1号梯5层flag" )
   END_RUNG
   RUNG wire#powerrail
      { S7_Templates := "SrcType := Byte" } EQ_Contact(in1 := "1号梯数据块"."1号梯当前楼层", in2 := 6)
      Coil( "1号梯数据块"."1号梯6层flag" )
   END_RUNG
   RUNG wire#powerrail
      { S7_Templates := "SrcType := Byte" } EQ_Contact(in1 := "1号梯数据块"."1号梯当前楼层", in2 := 7)
      Coil( "1号梯数据块"."1号梯7层flag" )
   END_RUNG
   RUNG wire#powerrail
      { S7_Templates := "SrcType := Byte" } EQ_Contact(in1 := "1号梯数据块"."1号梯当前楼层", in2 := 8)
      Coil( "1号梯数据块"."1号梯8层flag" )
   END_RUNG
   RUNG wire#powerrail
      { S7_Templates := "SrcType := Byte" } EQ_Contact(in1 := "1号梯数据块"."1号梯当前楼层", in2 := 9)
      Coil( "1号梯数据块"."1号梯9层flag" )
   END_RUNG
   RUNG wire#powerrail
      { S7_Templates := "SrcType := Byte" } EQ_Contact(in1 := "1号梯数据块"."1号梯当前楼层", in2 := 10)
      Coil( "1号梯数据块"."1号梯10层flag" )
   END_RUNG
   // the same network as SCL:
   "1号梯数据块"."1号梯1层flag" := "1号梯数据块"."1号梯当前楼层" = 1;
   "1号梯数据块"."1号梯2层flag" := "1号梯数据块"."1号梯当前楼层" = 2;
   "1号梯数据块"."1号梯3层flag" := "1号梯数据块"."1号梯当前楼层" = 3;
   "1号梯数据块"."1号梯4层flag" := "1号梯数据块"."1号梯当前楼层" = 4;
   "1号梯数据块"."1号梯5层flag" := "1号梯数据块"."1号梯当前楼层" = 5;
   "1号梯数据块"."1号梯6层flag" := "1号梯数据块"."1号梯当前楼层" = 6;
   "1号梯数据块"."1号梯7层flag" := "1号梯数据块"."1号梯当前楼层" = 7;
   "1号梯数据块"."1号梯8层flag" := "1号梯数据块"."1号梯当前楼层" = 8;
   "1号梯数据块"."1号梯9层flag" := "1号梯数据块"."1号梯当前楼层" = 9;
   "1号梯数据块"."1号梯10层flag" := "1号梯数据块"."1号梯当前楼层" = 10;
END_REGION

REGION Network 2: 1号梯楼层led_a显示
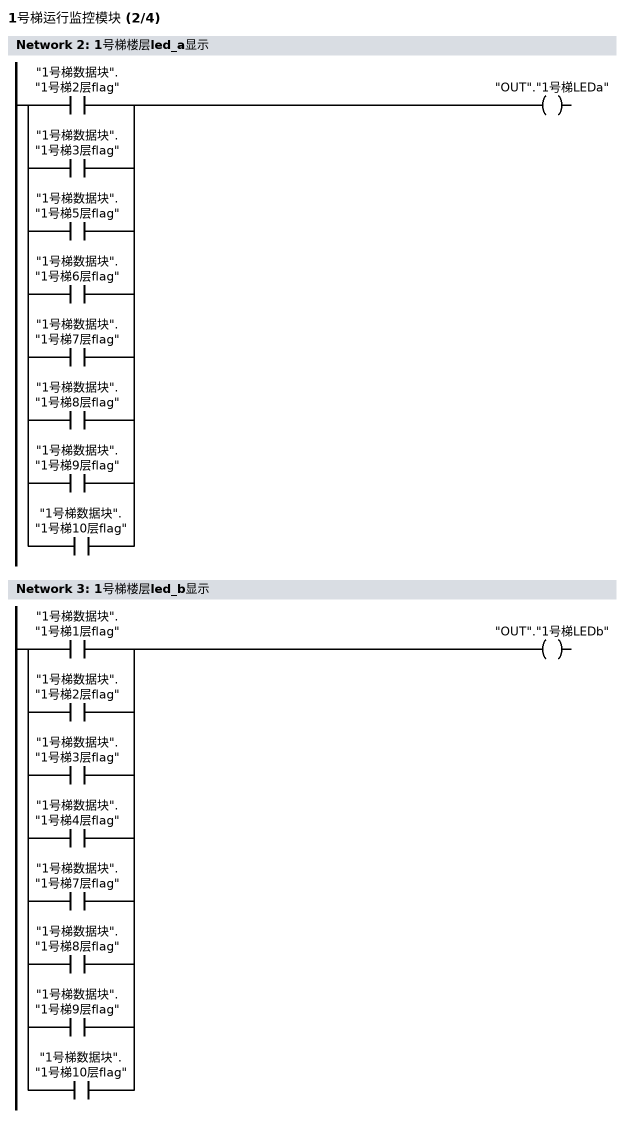
   RUNG wire#powerrail
      Contact( "1号梯数据块"."1号梯2层flag" )
      wire#w1
      Coil( "OUT"."1号梯LEDa" )
   END_RUNG
   RUNG wire#powerrail
      Contact( "1号梯数据块"."1号梯3层flag" )
   END_RUNG wire#w1
   RUNG wire#powerrail
      Contact( "1号梯数据块"."1号梯5层flag" )
   END_RUNG wire#w1
   RUNG wire#powerrail
      Contact( "1号梯数据块"."1号梯6层flag" )
   END_RUNG wire#w1
   RUNG wire#powerrail
      Contact( "1号梯数据块"."1号梯7层flag" )
   END_RUNG wire#w1
   RUNG wire#powerrail
      Contact( "1号梯数据块"."1号梯8层flag" )
   END_RUNG wire#w1
   RUNG wire#powerrail
      Contact( "1号梯数据块"."1号梯9层flag" )
   END_RUNG wire#w1
   RUNG wire#powerrail
      Contact( "1号梯数据块"."1号梯10层flag" )
   END_RUNG wire#w1
   // the same network as SCL:
   "OUT"."1号梯LEDa" := "1号梯数据块"."1号梯2层flag" OR "1号梯数据块"."1号梯3层flag" OR "1号梯数据块"."1号梯5层flag" OR "1号梯数据块"."1号梯6层flag" OR "1号梯数据块"."1号梯7层flag" OR "1号梯数据块"."1号梯8层flag" OR "1号梯数据块"."1号梯9层flag" OR "1号梯数据块"."1号梯10层flag";
END_REGION

REGION Network 3: 1号梯楼层led_b显示
   RUNG wire#powerrail
      Contact( "1号梯数据块"."1号梯1层flag" )
      wire#w1
      Coil( "OUT"."1号梯LEDb" )
   END_RUNG
   RUNG wire#powerrail
      Contact( "1号梯数据块"."1号梯2层flag" )
   END_RUNG wire#w1
   RUNG wire#powerrail
      Contact( "1号梯数据块"."1号梯3层flag" )
   END_RUNG wire#w1
   RUNG wire#powerrail
      Contact( "1号梯数据块"."1号梯4层flag" )
   END_RUNG wire#w1
   RUNG wire#powerrail
      Contact( "1号梯数据块"."1号梯7层flag" )
   END_RUNG wire#w1
   RUNG wire#powerrail
      Contact( "1号梯数据块"."1号梯8层flag" )
   END_RUNG wire#w1
   RUNG wire#powerrail
      Contact( "1号梯数据块"."1号梯9层flag" )
   END_RUNG wire#w1
   RUNG wire#powerrail
      Contact( "1号梯数据块"."1号梯10层flag" )
   END_RUNG wire#w1
   // the same network as SCL:
   "OUT"."1号梯LEDb" := "1号梯数据块"."1号梯1层flag" OR "1号梯数据块"."1号梯2层flag" OR "1号梯数据块"."1号梯3层flag" OR "1号梯数据块"."1号梯4层flag" OR "1号梯数据块"."1号梯7层flag" OR "1号梯数据块"."1号梯8层flag" OR "1号梯数据块"."1号梯9层flag" OR "1号梯数据块"."1号梯10层flag";
END_REGION

REGION Network 4: 1号梯楼层led_c显示
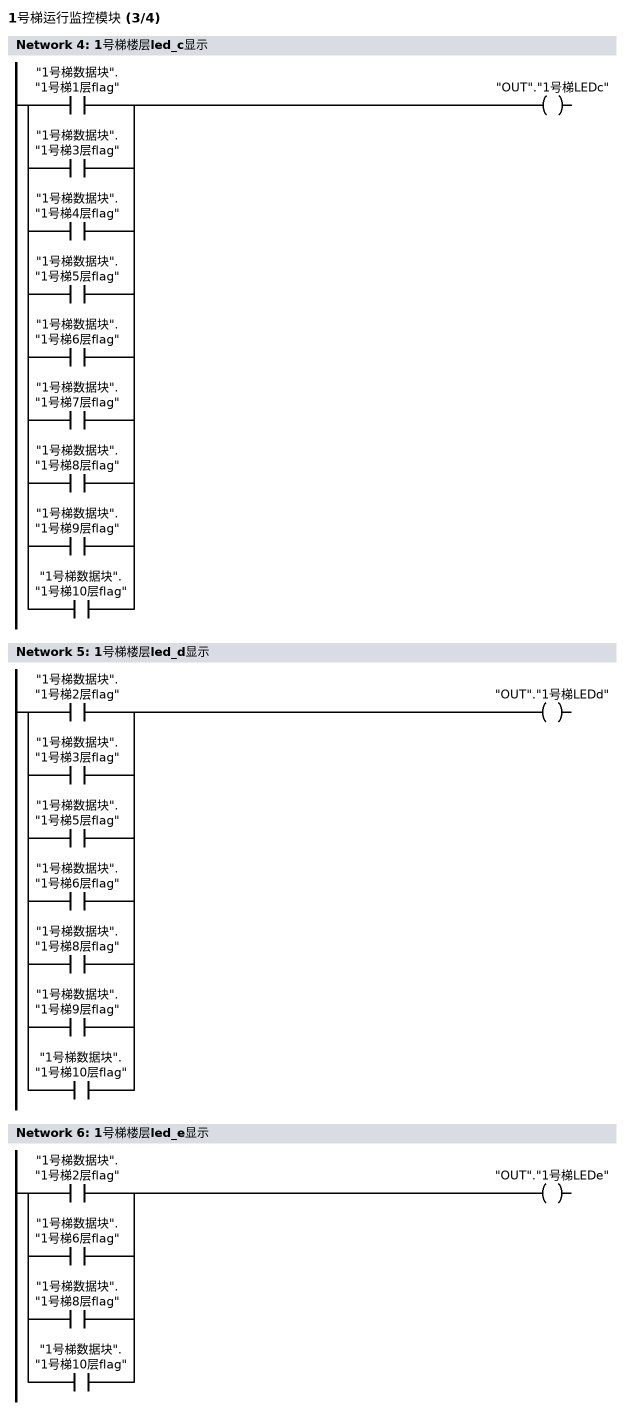
   RUNG wire#powerrail
      Contact( "1号梯数据块"."1号梯1层flag" )
      wire#w1
      Coil( "OUT"."1号梯LEDc" )
   END_RUNG
   RUNG wire#powerrail
      Contact( "1号梯数据块"."1号梯3层flag" )
   END_RUNG wire#w1
   RUNG wire#powerrail
      Contact( "1号梯数据块"."1号梯4层flag" )
   END_RUNG wire#w1
   RUNG wire#powerrail
      Contact( "1号梯数据块"."1号梯5层flag" )
   END_RUNG wire#w1
   RUNG wire#powerrail
      Contact( "1号梯数据块"."1号梯6层flag" )
   END_RUNG wire#w1
   RUNG wire#powerrail
      Contact( "1号梯数据块"."1号梯7层flag" )
   END_RUNG wire#w1
   RUNG wire#powerrail
      Contact( "1号梯数据块"."1号梯8层flag" )
   END_RUNG wire#w1
   RUNG wire#powerrail
      Contact( "1号梯数据块"."1号梯9层flag" )
   END_RUNG wire#w1
   RUNG wire#powerrail
      Contact( "1号梯数据块"."1号梯10层flag" )
   END_RUNG wire#w1
   // the same network as SCL:
   "OUT"."1号梯LEDc" := "1号梯数据块"."1号梯1层flag" OR "1号梯数据块"."1号梯3层flag" OR "1号梯数据块"."1号梯4层flag" OR "1号梯数据块"."1号梯5层flag" OR "1号梯数据块"."1号梯6层flag" OR "1号梯数据块"."1号梯7层flag" OR "1号梯数据块"."1号梯8层flag" OR "1号梯数据块"."1号梯9层flag" OR "1号梯数据块"."1号梯10层flag";
END_REGION

REGION Network 5: 1号梯楼层led_d显示
   RUNG wire#powerrail
      Contact( "1号梯数据块"."1号梯2层flag" )
      wire#w1
      Coil( "OUT"."1号梯LEDd" )
   END_RUNG
   RUNG wire#powerrail
      Contact( "1号梯数据块"."1号梯3层flag" )
   END_RUNG wire#w1
   RUNG wire#powerrail
      Contact( "1号梯数据块"."1号梯5层flag" )
   END_RUNG wire#w1
   RUNG wire#powerrail
      Contact( "1号梯数据块"."1号梯6层flag" )
   END_RUNG wire#w1
   RUNG wire#powerrail
      Contact( "1号梯数据块"."1号梯8层flag" )
   END_RUNG wire#w1
   RUNG wire#powerrail
      Contact( "1号梯数据块"."1号梯9层flag" )
   END_RUNG wire#w1
   RUNG wire#powerrail
      Contact( "1号梯数据块"."1号梯10层flag" )
   END_RUNG wire#w1
   // the same network as SCL:
   "OUT"."1号梯LEDd" := "1号梯数据块"."1号梯2层flag" OR "1号梯数据块"."1号梯3层flag" OR "1号梯数据块"."1号梯5层flag" OR "1号梯数据块"."1号梯6层flag" OR "1号梯数据块"."1号梯8层flag" OR "1号梯数据块"."1号梯9层flag" OR "1号梯数据块"."1号梯10层flag";
END_REGION

REGION Network 6: 1号梯楼层led_e显示
   RUNG wire#powerrail
      Contact( "1号梯数据块"."1号梯2层flag" )
      wire#w1
      Coil( "OUT"."1号梯LEDe" )
   END_RUNG
   RUNG wire#powerrail
      Contact( "1号梯数据块"."1号梯6层flag" )
   END_RUNG wire#w1
   RUNG wire#powerrail
      Contact( "1号梯数据块"."1号梯8层flag" )
   END_RUNG wire#w1
   RUNG wire#powerrail
      Contact( "1号梯数据块"."1号梯10层flag" )
   END_RUNG wire#w1
   // the same network as SCL:
   "OUT"."1号梯LEDe" := "1号梯数据块"."1号梯2层flag" OR "1号梯数据块"."1号梯6层flag" OR "1号梯数据块"."1号梯8层flag" OR "1号梯数据块"."1号梯10层flag";
END_REGION

REGION Network 7: 1号梯楼层led_f显示
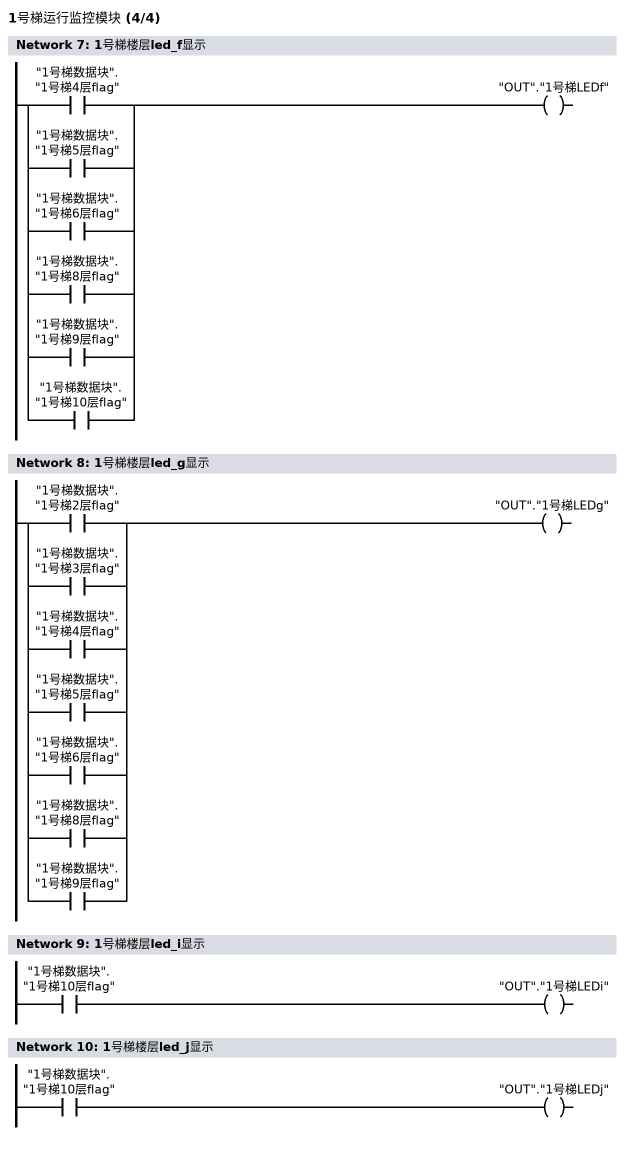
   RUNG wire#powerrail
      Contact( "1号梯数据块"."1号梯4层flag" )
      wire#w1
      Coil( "OUT"."1号梯LEDf" )
   END_RUNG
   RUNG wire#powerrail
      Contact( "1号梯数据块"."1号梯5层flag" )
   END_RUNG wire#w1
   RUNG wire#powerrail
      Contact( "1号梯数据块"."1号梯6层flag" )
   END_RUNG wire#w1
   RUNG wire#powerrail
      Contact( "1号梯数据块"."1号梯8层flag" )
   END_RUNG wire#w1
   RUNG wire#powerrail
      Contact( "1号梯数据块"."1号梯9层flag" )
   END_RUNG wire#w1
   RUNG wire#powerrail
      Contact( "1号梯数据块"."1号梯10层flag" )
   END_RUNG wire#w1
   // the same network as SCL:
   "OUT"."1号梯LEDf" := "1号梯数据块"."1号梯4层flag" OR "1号梯数据块"."1号梯5层flag" OR "1号梯数据块"."1号梯6层flag" OR "1号梯数据块"."1号梯8层flag" OR "1号梯数据块"."1号梯9层flag" OR "1号梯数据块"."1号梯10层flag";
END_REGION

REGION Network 8: 1号梯楼层led_g显示
   RUNG wire#powerrail
      Contact( "1号梯数据块"."1号梯2层flag" )
      wire#w1
      Coil( "OUT"."1号梯LEDg" )
   END_RUNG
   RUNG wire#powerrail
      Contact( "1号梯数据块"."1号梯3层flag" )
   END_RUNG wire#w1
   RUNG wire#powerrail
      Contact( "1号梯数据块"."1号梯4层flag" )
   END_RUNG wire#w1
   RUNG wire#powerrail
      Contact( "1号梯数据块"."1号梯5层flag" )
   END_RUNG wire#w1
   RUNG wire#powerrail
      Contact( "1号梯数据块"."1号梯6层flag" )
   END_RUNG wire#w1
   RUNG wire#powerrail
      Contact( "1号梯数据块"."1号梯8层flag" )
   END_RUNG wire#w1
   RUNG wire#powerrail
      Contact( "1号梯数据块"."1号梯9层flag" )
   END_RUNG wire#w1
   // the same network as SCL:
   "OUT"."1号梯LEDg" := "1号梯数据块"."1号梯2层flag" OR "1号梯数据块"."1号梯3层flag" OR "1号梯数据块"."1号梯4层flag" OR "1号梯数据块"."1号梯5层flag" OR "1号梯数据块"."1号梯6层flag" OR "1号梯数据块"."1号梯8层flag" OR "1号梯数据块"."1号梯9层flag";
END_REGION

REGION Network 9: 1号梯楼层led_i显示
   RUNG wire#powerrail
      Contact( "1号梯数据块"."1号梯10层flag" )
      Coil( "OUT"."1号梯LEDi" )
   END_RUNG
   // the same network as SCL:
   "OUT"."1号梯LEDi" := "1号梯数据块"."1号梯10层flag";
END_REGION

REGION Network 10: 1号梯楼层led_j显示
   RUNG wire#powerrail
      Contact( "1号梯数据块"."1号梯10层flag" )
      Coil( "OUT"."1号梯LEDj" )
   END_RUNG
   // the same network as SCL:
   "OUT"."1号梯LEDj" := "1号梯数据块"."1号梯10层flag";
END_REGION
END_FUNCTION

FUNCTION "1号梯启停控制" : Void   // FC20, LAD
{ S7_Optimized_Access := 'TRUE' }
VERSION : 0.1
   VAR_TEMP   // added for the SCL form of the ladder/FBD networks
      _w1 : Bool;
      _w2 : Bool;
   END_VAR
BEGIN

REGION Network 1: 1号梯开车判断
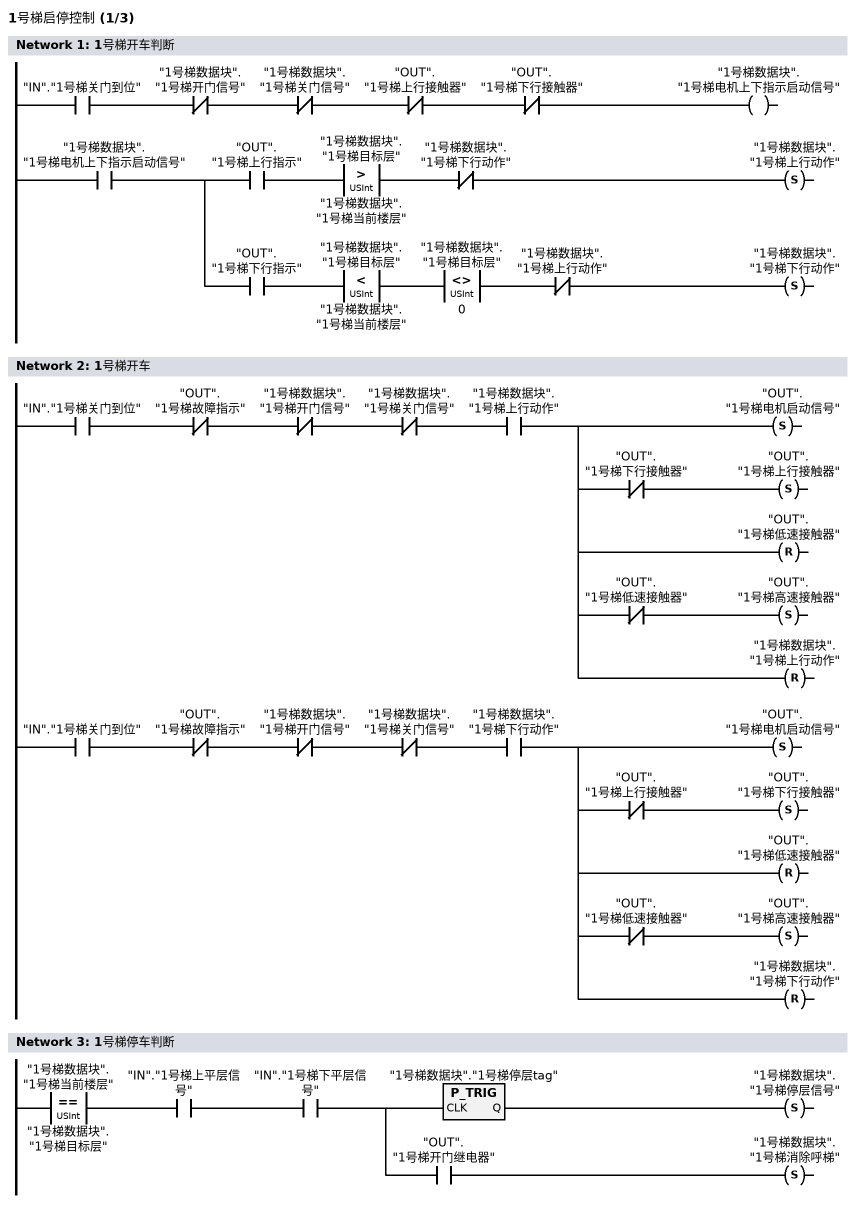
   RUNG wire#powerrail
      Contact( "IN"."1号梯关门到位" )
      I_Contact( "1号梯数据块"."1号梯开门信号" )
      I_Contact( "1号梯数据块"."1号梯关门信号" )
      I_Contact( "OUT"."1号梯上行接触器" )
      I_Contact( "OUT"."1号梯下行接触器" )
      Coil( "1号梯数据块"."1号梯电机上下指示启动信号" )
   END_RUNG
   RUNG wire#powerrail
      Contact( "1号梯数据块"."1号梯电机上下指示启动信号" )
      wire#w1
      Contact( "OUT"."1号梯上行指示" )
      { S7_Templates := "SrcType := USInt" } GT_Contact(in1 := "1号梯数据块"."1号梯目标层", in2 := "1号梯数据块"."1号梯当前楼层")
      I_Contact( "1号梯数据块"."1号梯下行动作" )
      S_Coil( "1号梯数据块"."1号梯上行动作" )
   END_RUNG
   RUNG wire#w1
      Contact( "OUT"."1号梯下行指示" )
      { S7_Templates := "SrcType := USInt" } LT_Contact(in1 := "1号梯数据块"."1号梯目标层", in2 := "1号梯数据块"."1号梯当前楼层")
      { S7_Templates := "SrcType := USInt" } NE_Contact(in1 := "1号梯数据块"."1号梯目标层", in2 := 0)
      I_Contact( "1号梯数据块"."1号梯上行动作" )
      S_Coil( "1号梯数据块"."1号梯下行动作" )
   END_RUNG
   // the same network as SCL:
   "1号梯数据块"."1号梯电机上下指示启动信号" := "IN"."1号梯关门到位" AND NOT "1号梯数据块"."1号梯开门信号" AND NOT "1号梯数据块"."1号梯关门信号" AND NOT "OUT"."1号梯上行接触器" AND NOT "OUT"."1号梯下行接触器";
   IF "1号梯数据块"."1号梯电机上下指示启动信号" AND "OUT"."1号梯上行指示" AND ("1号梯数据块"."1号梯目标层" > "1号梯数据块"."1号梯当前楼层") AND NOT "1号梯数据块"."1号梯下行动作" THEN
       "1号梯数据块"."1号梯上行动作" := TRUE;
   END_IF;
   IF "1号梯数据块"."1号梯电机上下指示启动信号" AND "OUT"."1号梯下行指示" AND ("1号梯数据块"."1号梯目标层" < "1号梯数据块"."1号梯当前楼层") AND ("1号梯数据块"."1号梯目标层" <> 0) AND NOT "1号梯数据块"."1号梯上行动作" THEN
       "1号梯数据块"."1号梯下行动作" := TRUE;
   END_IF;
END_REGION

REGION Network 2: 1号梯开车
   RUNG wire#powerrail
      Contact( "IN"."1号梯关门到位" )
      I_Contact( "OUT"."1号梯故障指示" )
      I_Contact( "1号梯数据块"."1号梯开门信号" )
      I_Contact( "1号梯数据块"."1号梯关门信号" )
      Contact( "1号梯数据块"."1号梯上行动作" )
      wire#w1
      S_Coil( "OUT"."1号梯电机启动信号" )
   END_RUNG
   RUNG wire#w1
      I_Contact( "OUT"."1号梯下行接触器" )
      S_Coil( "OUT"."1号梯上行接触器" )
   END_RUNG
   RUNG wire#w1
      R_Coil( "OUT"."1号梯低速接触器" )
   END_RUNG
   RUNG wire#w1
      I_Contact( "OUT"."1号梯低速接触器" )
      S_Coil( "OUT"."1号梯高速接触器" )
   END_RUNG
   RUNG wire#w1
      R_Coil( "1号梯数据块"."1号梯上行动作" )
   END_RUNG
   RUNG wire#powerrail
      Contact( "IN"."1号梯关门到位" )
      I_Contact( "OUT"."1号梯故障指示" )
      I_Contact( "1号梯数据块"."1号梯开门信号" )
      I_Contact( "1号梯数据块"."1号梯关门信号" )
      Contact( "1号梯数据块"."1号梯下行动作" )
      wire#w2
      S_Coil( "OUT"."1号梯电机启动信号" )
   END_RUNG
   RUNG wire#w2
      I_Contact( "OUT"."1号梯上行接触器" )
      S_Coil( "OUT"."1号梯下行接触器" )
   END_RUNG
   RUNG wire#w2
      R_Coil( "OUT"."1号梯低速接触器" )
   END_RUNG
   RUNG wire#w2
      I_Contact( "OUT"."1号梯低速接触器" )
      S_Coil( "OUT"."1号梯高速接触器" )
   END_RUNG
   RUNG wire#w2
      R_Coil( "1号梯数据块"."1号梯下行动作" )
   END_RUNG
   // the same network as SCL:
   #_w1 := "IN"."1号梯关门到位" AND NOT "OUT"."1号梯故障指示" AND NOT "1号梯数据块"."1号梯开门信号" AND NOT "1号梯数据块"."1号梯关门信号" AND "1号梯数据块"."1号梯上行动作";
   IF #_w1 THEN "OUT"."1号梯电机启动信号" := TRUE; END_IF;
   IF #_w1 AND NOT "OUT"."1号梯下行接触器" THEN "OUT"."1号梯上行接触器" := TRUE; END_IF;
   IF #_w1 THEN "OUT"."1号梯低速接触器" := FALSE; END_IF;
   IF #_w1 AND NOT "OUT"."1号梯低速接触器" THEN "OUT"."1号梯高速接触器" := TRUE; END_IF;
   IF #_w1 THEN "1号梯数据块"."1号梯上行动作" := FALSE; END_IF;
   #_w2 := "IN"."1号梯关门到位" AND NOT "OUT"."1号梯故障指示" AND NOT "1号梯数据块"."1号梯开门信号" AND NOT "1号梯数据块"."1号梯关门信号" AND "1号梯数据块"."1号梯下行动作";
   IF #_w2 THEN "OUT"."1号梯电机启动信号" := TRUE; END_IF;
   IF #_w2 AND NOT "OUT"."1号梯上行接触器" THEN "OUT"."1号梯下行接触器" := TRUE; END_IF;
   IF #_w2 THEN "OUT"."1号梯低速接触器" := FALSE; END_IF;
   IF #_w2 AND NOT "OUT"."1号梯低速接触器" THEN "OUT"."1号梯高速接触器" := TRUE; END_IF;
   IF #_w2 THEN "1号梯数据块"."1号梯下行动作" := FALSE; END_IF;
END_REGION

REGION Network 3: 1号梯停车判断
   RUNG wire#powerrail
      { S7_Templates := "SrcType := USInt" } EQ_Contact(in1 := "1号梯数据块"."1号梯当前楼层", in2 := "1号梯数据块"."1号梯目标层")
      Contact( "IN"."1号梯上平层信号" )
      Contact( "IN"."1号梯下平层信号" )
      wire#w1
      P_Trig( "1号梯数据块"."1号梯停层tag" )
      S_Coil( "1号梯数据块"."1号梯停层信号" )
   END_RUNG
   RUNG wire#w1
      Contact( "OUT"."1号梯开门继电器" )
      S_Coil( "1号梯数据块"."1号梯消除呼梯" )
   END_RUNG
   // the same network as SCL:
   #_w1 := ("1号梯数据块"."1号梯当前楼层" = "1号梯数据块"."1号梯目标层") AND "IN"."1号梯上平层信号" AND "IN"."1号梯下平层信号";
   #_w2 := #_w1 AND NOT "1号梯数据块"."1号梯停层tag";   // rising edge
   "1号梯数据块"."1号梯停层tag" := #_w1;
   IF #_w2 THEN "1号梯数据块"."1号梯停层信号" := TRUE; END_IF;
   IF #_w1 AND "OUT"."1号梯开门继电器" THEN "1号梯数据块"."1号梯消除呼梯" := TRUE; END_IF;
END_REGION

REGION Network 4: 1号梯三级制动
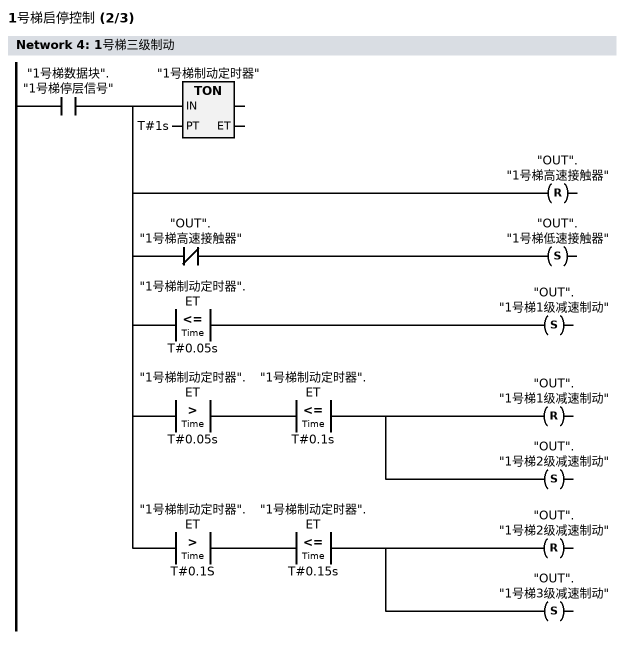
   "1号梯制动定时器".TON(IN := "1号梯数据块"."1号梯停层信号", PT := T#1s);
   IF "1号梯数据块"."1号梯停层信号" THEN "OUT"."1号梯高速接触器" := FALSE; END_IF;
   IF "1号梯数据块"."1号梯停层信号" AND NOT "OUT"."1号梯高速接触器" THEN "OUT"."1号梯低速接触器" := TRUE; END_IF;
   IF "1号梯数据块"."1号梯停层信号" AND ("1号梯制动定时器".ET <= T#0.05s) THEN "OUT"."1号梯1级减速制动" := TRUE; END_IF;
   IF "1号梯数据块"."1号梯停层信号" AND ("1号梯制动定时器".ET > T#0.05s) AND ("1号梯制动定时器".ET <= T#0.1s) THEN
       "OUT"."1号梯1级减速制动" := FALSE;
       "OUT"."1号梯2级减速制动" := TRUE;
   END_IF;
   IF "1号梯数据块"."1号梯停层信号" AND ("1号梯制动定时器".ET > T#0.1S) AND ("1号梯制动定时器".ET <= T#0.15s) THEN
       "OUT"."1号梯2级减速制动" := FALSE;
       "OUT"."1号梯3级减速制动" := TRUE;
   END_IF;
END_REGION

REGION Network 5: 1号梯停车与检修停车（消除呼梯）
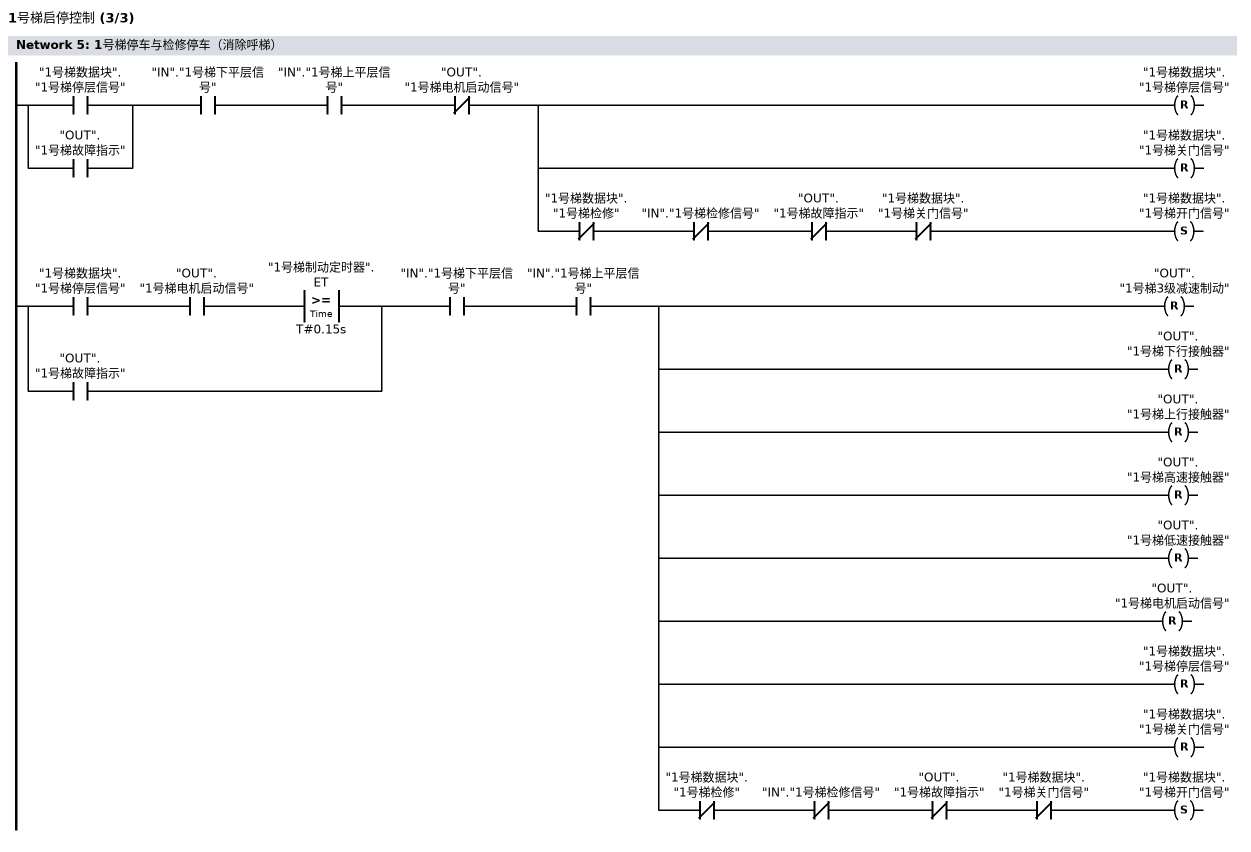
   RUNG wire#powerrail
      Contact( "1号梯数据块"."1号梯停层信号" )
      wire#w1
      Contact( "IN"."1号梯下平层信号" )
      Contact( "IN"."1号梯上平层信号" )
      I_Contact( "OUT"."1号梯电机启动信号" )
      wire#w2
      R_Coil( "1号梯数据块"."1号梯停层信号" )
   END_RUNG
   RUNG wire#powerrail
      Contact( "OUT"."1号梯故障指示" )
   END_RUNG wire#w1
   RUNG wire#w2
      R_Coil( "1号梯数据块"."1号梯关门信号" )
   END_RUNG
   RUNG wire#w2
      I_Contact( "1号梯数据块"."1号梯检修" )
      I_Contact( "IN"."1号梯检修信号" )
      I_Contact( "OUT"."1号梯故障指示" )
      I_Contact( "1号梯数据块"."1号梯关门信号" )
      S_Coil( "1号梯数据块"."1号梯开门信号" )
   END_RUNG
   RUNG wire#powerrail
      Contact( "1号梯数据块"."1号梯停层信号" )
      Contact( "OUT"."1号梯电机启动信号" )
      { S7_Templates := "SrcType := Time" } GE_Contact(in1 := "1号梯制动定时器".ET, in2 := T#0.15s)
      wire#w3
      Contact( "IN"."1号梯下平层信号" )
      Contact( "IN"."1号梯上平层信号" )
      wire#w4
      R_Coil( "OUT"."1号梯3级减速制动" )
   END_RUNG
   RUNG wire#powerrail
      Contact( "OUT"."1号梯故障指示" )
   END_RUNG wire#w3
   RUNG wire#w4
      R_Coil( "OUT"."1号梯下行接触器" )
   END_RUNG
   RUNG wire#w4
      R_Coil( "OUT"."1号梯上行接触器" )
   END_RUNG
   RUNG wire#w4
      R_Coil( "OUT"."1号梯高速接触器" )
   END_RUNG
   RUNG wire#w4
      R_Coil( "OUT"."1号梯低速接触器" )
   END_RUNG
   RUNG wire#w4
      R_Coil( "OUT"."1号梯电机启动信号" )
   END_RUNG
   RUNG wire#w4
      R_Coil( "1号梯数据块"."1号梯停层信号" )
   END_RUNG
   RUNG wire#w4
      R_Coil( "1号梯数据块"."1号梯关门信号" )
   END_RUNG
   RUNG wire#w4
      I_Contact( "1号梯数据块"."1号梯检修" )
      I_Contact( "IN"."1号梯检修信号" )
      I_Contact( "OUT"."1号梯故障指示" )
      I_Contact( "1号梯数据块"."1号梯关门信号" )
      S_Coil( "1号梯数据块"."1号梯开门信号" )
   END_RUNG
   // the same network as SCL:
   #_w1 := ("1号梯数据块"."1号梯停层信号" OR "OUT"."1号梯故障指示") AND "IN"."1号梯下平层信号" AND "IN"."1号梯上平层信号" AND NOT "OUT"."1号梯电机启动信号";
   IF #_w1 THEN
       "1号梯数据块"."1号梯停层信号" := FALSE;
       "1号梯数据块"."1号梯关门信号" := FALSE;
   END_IF;
   IF #_w1 AND NOT "1号梯数据块"."1号梯检修" AND NOT "IN"."1号梯检修信号" AND NOT "OUT"."1号梯故障指示" AND NOT "1号梯数据块"."1号梯关门信号" THEN
       "1号梯数据块"."1号梯开门信号" := TRUE;
   END_IF;
   #_w2 := (("1号梯数据块"."1号梯停层信号" AND "OUT"."1号梯电机启动信号" AND ("1号梯制动定时器".ET >= T#0.15s)) OR "OUT"."1号梯故障指示") AND "IN"."1号梯下平层信号" AND "IN"."1号梯上平层信号";
   IF #_w2 THEN
       "OUT"."1号梯3级减速制动" := FALSE;
       "OUT"."1号梯下行接触器" := FALSE;
       "OUT"."1号梯上行接触器" := FALSE;
       "OUT"."1号梯高速接触器" := FALSE;
       "OUT"."1号梯低速接触器" := FALSE;
       "OUT"."1号梯电机启动信号" := FALSE;
       "1号梯数据块"."1号梯停层信号" := FALSE;
       "1号梯数据块"."1号梯关门信号" := FALSE;
   END_IF;
   IF #_w2 AND NOT "1号梯数据块"."1号梯检修" AND NOT "IN"."1号梯检修信号" AND NOT "OUT"."1号梯故障指示" AND NOT "1号梯数据块"."1号梯关门信号" THEN
       "1号梯数据块"."1号梯开门信号" := TRUE;
   END_IF;
END_REGION
END_FUNCTION

FUNCTION "1号梯开关门控制" : Void   // FC26, LAD
{ S7_Optimized_Access := 'TRUE' }
VERSION : 0.1
   VAR_TEMP   // added for the SCL form of the ladder/FBD networks
      _w1 : Bool;
      _w2 : Bool;
   END_VAR
BEGIN

REGION Network 1: 1号梯双平层信号
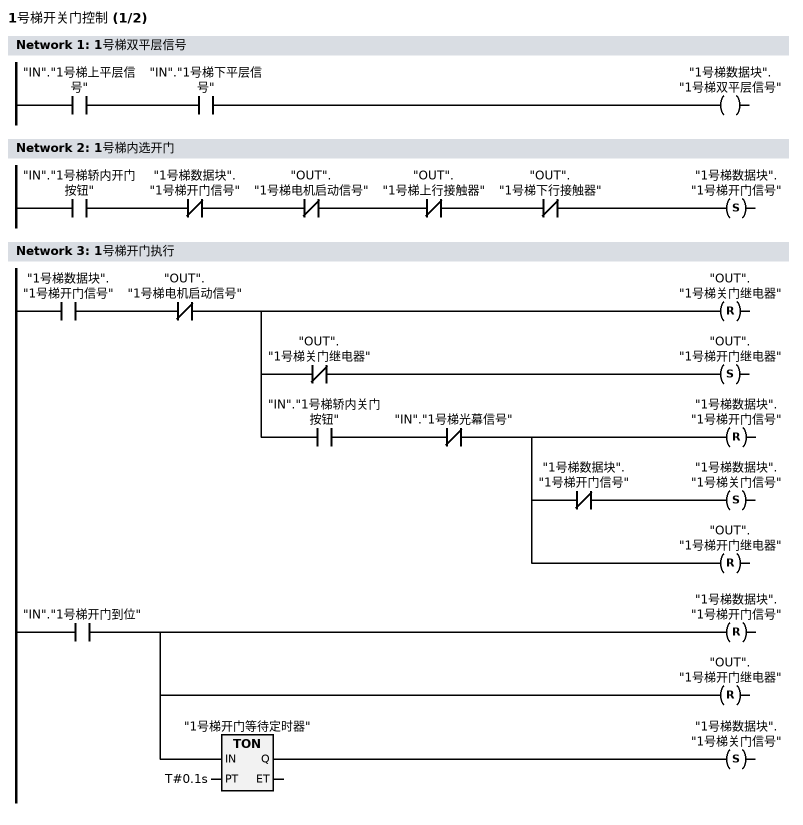
   RUNG wire#powerrail
      Contact( "IN"."1号梯上平层信号" )
      Contact( "IN"."1号梯下平层信号" )
      Coil( "1号梯数据块"."1号梯双平层信号" )
   END_RUNG
   // the same network as SCL:
   "1号梯数据块"."1号梯双平层信号" := "IN"."1号梯上平层信号" AND "IN"."1号梯下平层信号";
END_REGION

REGION Network 2: 1号梯内选开门
   RUNG wire#powerrail
      Contact( "IN"."1号梯轿内开门按钮" )
      I_Contact( "1号梯数据块"."1号梯开门信号" )
      I_Contact( "OUT"."1号梯电机启动信号" )
      I_Contact( "OUT"."1号梯上行接触器" )
      I_Contact( "OUT"."1号梯下行接触器" )
      S_Coil( "1号梯数据块"."1号梯开门信号" )
   END_RUNG
   // the same network as SCL:
   IF "IN"."1号梯轿内开门按钮" AND NOT "1号梯数据块"."1号梯开门信号" AND NOT "OUT"."1号梯电机启动信号" AND NOT "OUT"."1号梯上行接触器" AND NOT "OUT"."1号梯下行接触器" THEN
       "1号梯数据块"."1号梯开门信号" := TRUE;
   END_IF;
END_REGION

REGION Network 3: 1号梯开门执行
   #_w1 := "1号梯数据块"."1号梯开门信号" AND NOT "OUT"."1号梯电机启动信号";
   IF #_w1 THEN "OUT"."1号梯关门继电器" := FALSE; END_IF;
   IF #_w1 AND NOT "OUT"."1号梯关门继电器" THEN "OUT"."1号梯开门继电器" := TRUE; END_IF;
   #_w2 := #_w1 AND "IN"."1号梯轿内关门按钮" AND NOT "IN"."1号梯光幕信号";
   IF #_w2 THEN "1号梯数据块"."1号梯开门信号" := FALSE; END_IF;
   IF #_w2 AND NOT "1号梯数据块"."1号梯开门信号" THEN "1号梯数据块"."1号梯关门信号" := TRUE; END_IF;
   IF #_w2 THEN "OUT"."1号梯开门继电器" := FALSE; END_IF;
   IF "IN"."1号梯开门到位" THEN
       "1号梯数据块"."1号梯开门信号" := FALSE;
       "OUT"."1号梯开门继电器" := FALSE;
   END_IF;
   "1号梯开门等待定时器".TON(IN := "IN"."1号梯开门到位", PT := T#0.1s);
   IF "1号梯开门等待定时器".Q THEN "1号梯数据块"."1号梯关门信号" := TRUE; END_IF;
END_REGION

REGION Network 4: 1号梯关门执行
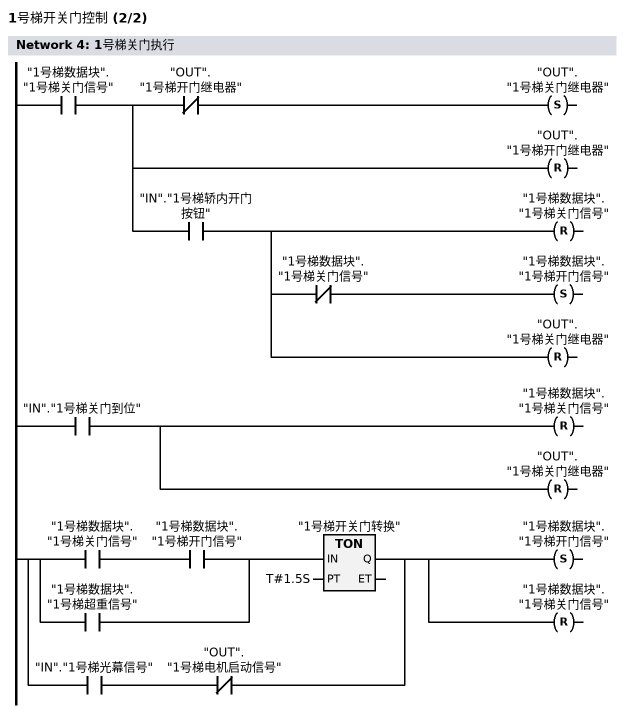
   IF "1号梯数据块"."1号梯关门信号" AND NOT "OUT"."1号梯开门继电器" THEN "OUT"."1号梯关门继电器" := TRUE; END_IF;
   IF "1号梯数据块"."1号梯关门信号" THEN "OUT"."1号梯开门继电器" := FALSE; END_IF;
   #_w1 := "1号梯数据块"."1号梯关门信号" AND "IN"."1号梯轿内开门按钮";
   IF #_w1 THEN "1号梯数据块"."1号梯关门信号" := FALSE; END_IF;
   IF #_w1 AND NOT "1号梯数据块"."1号梯关门信号" THEN "1号梯数据块"."1号梯开门信号" := TRUE; END_IF;
   IF #_w1 THEN "OUT"."1号梯关门继电器" := FALSE; END_IF;
   IF "IN"."1号梯关门到位" THEN
       "1号梯数据块"."1号梯关门信号" := FALSE;
       "OUT"."1号梯关门继电器" := FALSE;
   END_IF;
   "1号梯开关门转换".TON(IN := ("1号梯数据块"."1号梯关门信号" AND "1号梯数据块"."1号梯开门信号") OR "1号梯数据块"."1号梯超重信号", PT := T#1.5S);
   IF "1号梯开关门转换".Q OR ("IN"."1号梯光幕信号" AND NOT "OUT"."1号梯电机启动信号") THEN
       "1号梯数据块"."1号梯开门信号" := TRUE;
       "1号梯数据块"."1号梯关门信号" := FALSE;
   END_IF;
END_REGION
END_FUNCTION

FUNCTION "1号梯楼层计数" : Void   // FC32, LAD
{ S7_Optimized_Access := 'TRUE' }
VERSION : 0.1
   VAR_TEMP   // added for the SCL form of the ladder/FBD networks
      _w1 : Bool;
      _w2 : Bool;
   END_VAR
BEGIN

REGION Network 1: 1号梯楼层计数、楼层判断解码
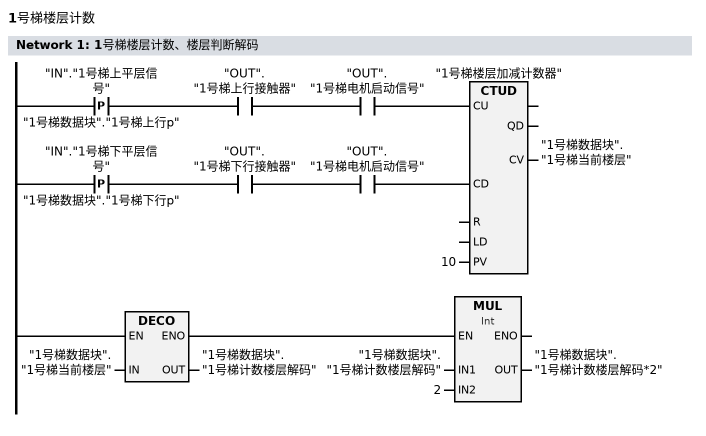
   #_w1 := "IN"."1号梯上平层信号" AND NOT "1号梯数据块"."1号梯上行p";   // rising edge of "IN"."1号梯上平层信号"
   "1号梯数据块"."1号梯上行p" := "IN"."1号梯上平层信号";
   #_w2 := "IN"."1号梯下平层信号" AND NOT "1号梯数据块"."1号梯下行p";   // rising edge of "IN"."1号梯下平层信号"
   "1号梯数据块"."1号梯下行p" := "IN"."1号梯下平层信号";
   "1号梯楼层加减计数器".CTUD(CU := #_w1 AND "OUT"."1号梯上行接触器" AND "OUT"."1号梯电机启动信号",
                     CD := #_w2 AND "OUT"."1号梯下行接触器" AND "OUT"."1号梯电机启动信号",
                     PV := 10,
                     CV => "1号梯数据块"."1号梯当前楼层");
   "1号梯数据块"."1号梯计数楼层解码" := DECO(IN := "1号梯数据块"."1号梯当前楼层");
   "1号梯数据块"."1号梯计数楼层解码*2" := "1号梯数据块"."1号梯计数楼层解码" * 2;
END_REGION
END_FUNCTION

FUNCTION "1号梯超重和内选" : Void   // FC39, LAD
{ S7_Optimized_Access := 'TRUE' }
VERSION : 0.1
BEGIN

REGION Network 1: 一号梯体重转换
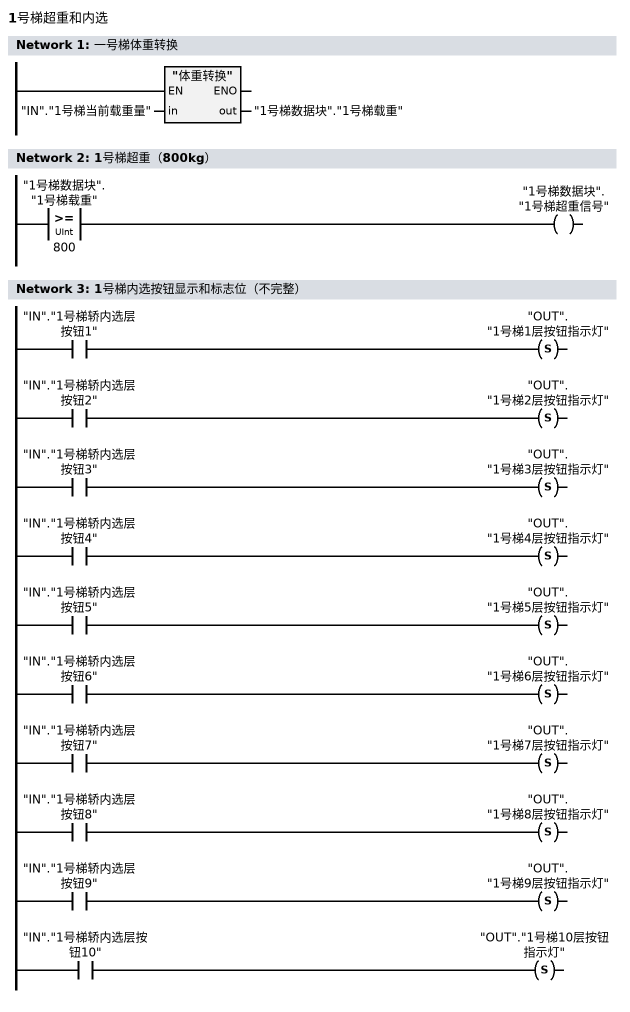
   RUNG wire#powerrail
      "体重转换"(in := "IN"."1号梯当前载重量", out => "1号梯数据块"."1号梯载重")
   END_RUNG
   // the same network as SCL:
   "体重转换"(in := "IN"."1号梯当前载重量", out => "1号梯数据块"."1号梯载重");
END_REGION

REGION Network 2: 1号梯超重（800kg）
   RUNG wire#powerrail
      { S7_Templates := "SrcType := UInt" } GE_Contact(in1 := "1号梯数据块"."1号梯载重", in2 := 800)
      Coil( "1号梯数据块"."1号梯超重信号" )
   END_RUNG
   // the same network as SCL:
   "1号梯数据块"."1号梯超重信号" := "1号梯数据块"."1号梯载重" >= 800;
END_REGION

REGION Network 3: 1号梯内选按钮显示和标志位（不完整）
   RUNG wire#powerrail
      Contact( "IN"."1号梯轿内选层按钮1" )
      S_Coil( "OUT"."1号梯1层按钮指示灯" )
   END_RUNG
   RUNG wire#powerrail
      Contact( "IN"."1号梯轿内选层按钮2" )
      S_Coil( "OUT"."1号梯2层按钮指示灯" )
   END_RUNG
   RUNG wire#powerrail
      Contact( "IN"."1号梯轿内选层按钮3" )
      S_Coil( "OUT"."1号梯3层按钮指示灯" )
   END_RUNG
   RUNG wire#powerrail
      Contact( "IN"."1号梯轿内选层按钮4" )
      S_Coil( "OUT"."1号梯4层按钮指示灯" )
   END_RUNG
   RUNG wire#powerrail
      Contact( "IN"."1号梯轿内选层按钮5" )
      S_Coil( "OUT"."1号梯5层按钮指示灯" )
   END_RUNG
   RUNG wire#powerrail
      Contact( "IN"."1号梯轿内选层按钮6" )
      S_Coil( "OUT"."1号梯6层按钮指示灯" )
   END_RUNG
   RUNG wire#powerrail
      Contact( "IN"."1号梯轿内选层按钮7" )
      S_Coil( "OUT"."1号梯7层按钮指示灯" )
   END_RUNG
   RUNG wire#powerrail
      Contact( "IN"."1号梯轿内选层按钮8" )
      S_Coil( "OUT"."1号梯8层按钮指示灯" )
   END_RUNG
   RUNG wire#powerrail
      Contact( "IN"."1号梯轿内选层按钮9" )
      S_Coil( "OUT"."1号梯9层按钮指示灯" )
   END_RUNG
   RUNG wire#powerrail
      Contact( "IN"."1号梯轿内选层按钮10" )
      S_Coil( "OUT"."1号梯10层按钮指示灯" )
   END_RUNG
   // the same network as SCL:
   IF "IN"."1号梯轿内选层按钮1" THEN "OUT"."1号梯1层按钮指示灯" := TRUE; END_IF;
   IF "IN"."1号梯轿内选层按钮2" THEN "OUT"."1号梯2层按钮指示灯" := TRUE; END_IF;
   IF "IN"."1号梯轿内选层按钮3" THEN "OUT"."1号梯3层按钮指示灯" := TRUE; END_IF;
   IF "IN"."1号梯轿内选层按钮4" THEN "OUT"."1号梯4层按钮指示灯" := TRUE; END_IF;
   IF "IN"."1号梯轿内选层按钮5" THEN "OUT"."1号梯5层按钮指示灯" := TRUE; END_IF;
   IF "IN"."1号梯轿内选层按钮6" THEN "OUT"."1号梯6层按钮指示灯" := TRUE; END_IF;
   IF "IN"."1号梯轿内选层按钮7" THEN "OUT"."1号梯7层按钮指示灯" := TRUE; END_IF;
   IF "IN"."1号梯轿内选层按钮8" THEN "OUT"."1号梯8层按钮指示灯" := TRUE; END_IF;
   IF "IN"."1号梯轿内选层按钮9" THEN "OUT"."1号梯9层按钮指示灯" := TRUE; END_IF;
   IF "IN"."1号梯轿内选层按钮10" THEN "OUT"."1号梯10层按钮指示灯" := TRUE; END_IF;
END_REGION
END_FUNCTION

FUNCTION "1号梯检修" : Void   // FC41, LAD
{ S7_Optimized_Access := 'TRUE' }
VERSION : 0.1
BEGIN
END_FUNCTION

FUNCTION "1号梯目标楼层与方向判断" : Void   // FC42, LAD
{ S7_Optimized_Access := 'TRUE' }
VERSION : 0.1
BEGIN
END_FUNCTION

FUNCTION "1号梯字节消除与记录" : Void   // FC43, LAD
{ S7_Optimized_Access := 'TRUE' }
VERSION : 0.1
BEGIN
END_FUNCTION

// folder: 2号梯

FUNCTION "2号梯初始化" : Void   // FC3, LAD
{ S7_Optimized_Access := 'TRUE' }
VERSION : 0.1
   VAR_INPUT
      初始化方向 : Bool;
      初始化楼层 : Byte;
   END_VAR
   VAR_TEMP   // added for the SCL form of the ladder/FBD networks
      _w1 : Bool;
      _w2 : Bool;
      _w3 : Bool;
      _w4 : Bool;
   END_VAR
BEGIN

REGION Network 1: 2号梯传参（方向+初始化楼层）
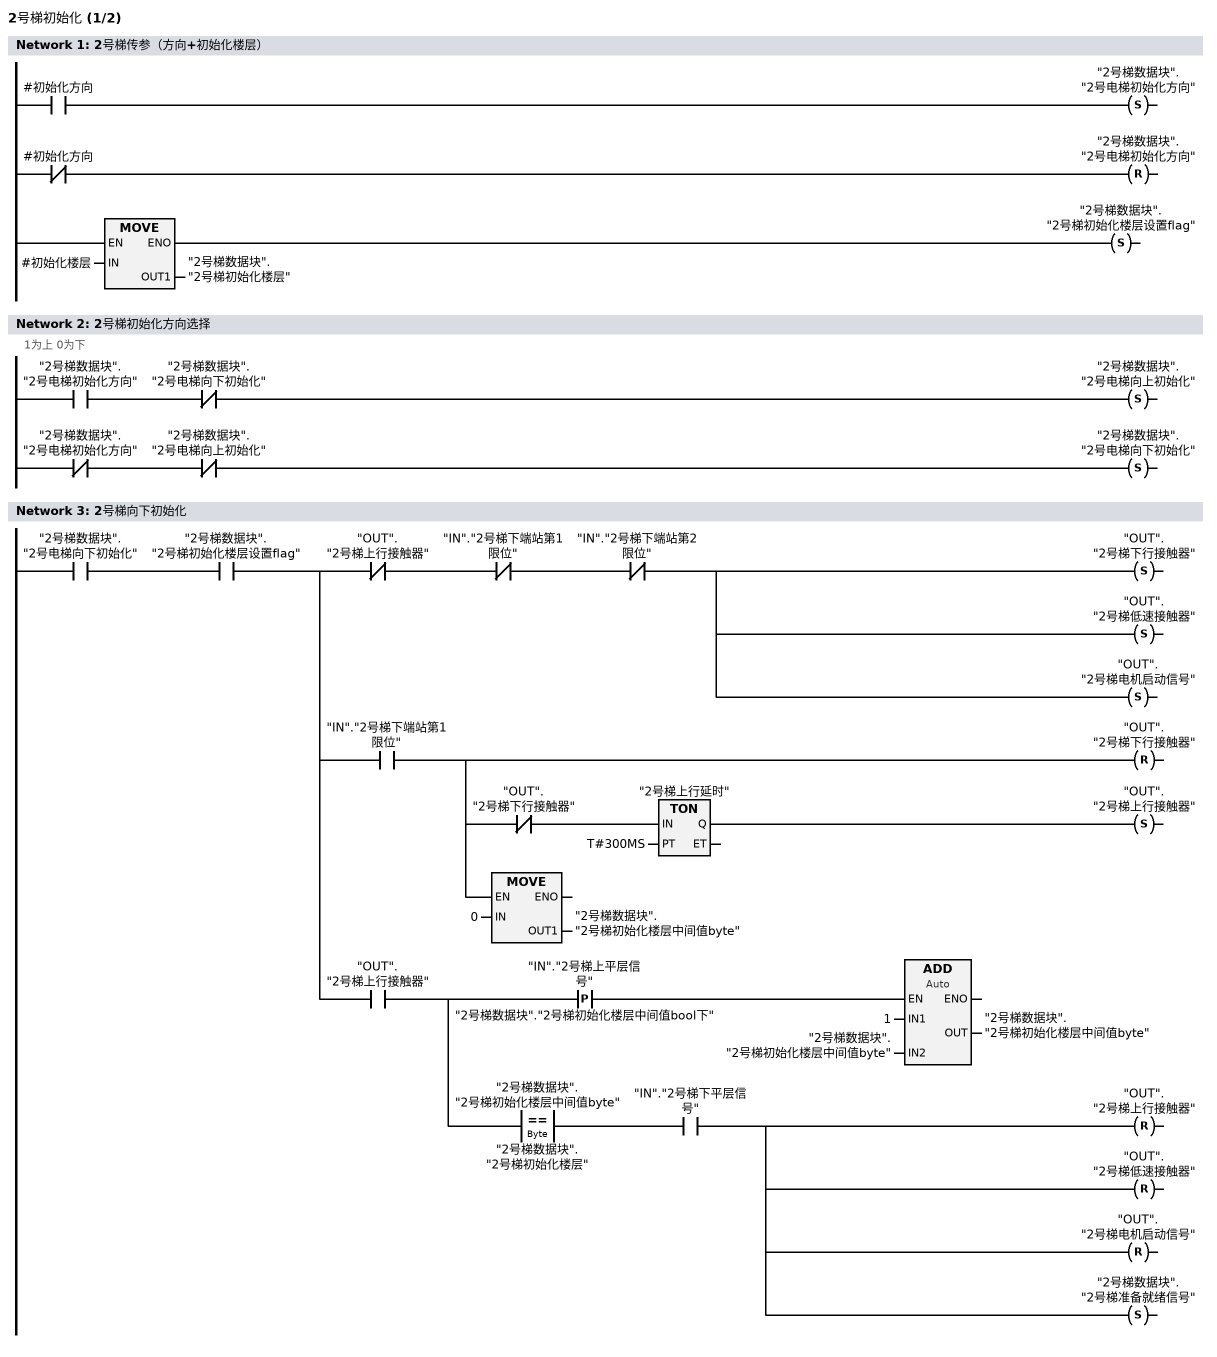
   RUNG wire#powerrail
      Contact( #初始化方向 )
      S_Coil( "2号梯数据块"."2号电梯初始化方向" )
   END_RUNG
   RUNG wire#powerrail
      I_Contact( #初始化方向 )
      R_Coil( "2号梯数据块"."2号电梯初始化方向" )
   END_RUNG
   RUNG wire#powerrail
      Move(in := #初始化楼层, out1 => "2号梯数据块"."2号梯初始化楼层")
      S_Coil( "2号梯数据块"."2号梯初始化楼层设置flag" )
   END_RUNG
   // the same network as SCL:
   IF #初始化方向 THEN "2号梯数据块"."2号电梯初始化方向" := TRUE; END_IF;
   IF NOT #初始化方向 THEN "2号梯数据块"."2号电梯初始化方向" := FALSE; END_IF;
   "2号梯数据块"."2号梯初始化楼层" := #初始化楼层;
   "2号梯数据块"."2号梯初始化楼层设置flag" := TRUE;
END_REGION

REGION Network 2: 2号梯初始化方向选择
   // 1为上 0为下
   RUNG wire#powerrail
      Contact( "2号梯数据块"."2号电梯初始化方向" )
      I_Contact( "2号梯数据块"."2号电梯向下初始化" )
      S_Coil( "2号梯数据块"."2号电梯向上初始化" )
   END_RUNG
   RUNG wire#powerrail
      I_Contact( "2号梯数据块"."2号电梯初始化方向" )
      I_Contact( "2号梯数据块"."2号电梯向上初始化" )
      S_Coil( "2号梯数据块"."2号电梯向下初始化" )
   END_RUNG
   // the same network as SCL:
   IF "2号梯数据块"."2号电梯初始化方向" AND NOT "2号梯数据块"."2号电梯向下初始化" THEN "2号梯数据块"."2号电梯向上初始化" := TRUE; END_IF;
   IF NOT "2号梯数据块"."2号电梯初始化方向" AND NOT "2号梯数据块"."2号电梯向上初始化" THEN "2号梯数据块"."2号电梯向下初始化" := TRUE; END_IF;
END_REGION

REGION Network 3: 2号梯向下初始化
   #_w1 := "2号梯数据块"."2号电梯向下初始化" AND "2号梯数据块"."2号梯初始化楼层设置flag";
   IF #_w1 AND NOT "OUT"."2号梯上行接触器" AND NOT "IN"."2号梯下端站第1限位" AND NOT "IN"."2号梯下端站第2限位" THEN
       "OUT"."2号梯下行接触器" := TRUE;
       "OUT"."2号梯低速接触器" := TRUE;
       "OUT"."2号梯电机启动信号" := TRUE;
   END_IF;
   #_w2 := #_w1 AND "IN"."2号梯下端站第1限位";
   IF #_w2 THEN "OUT"."2号梯下行接触器" := FALSE; END_IF;
   "2号梯上行延时".TON(IN := #_w2 AND NOT "OUT"."2号梯下行接触器", PT := T#300MS);
   IF "2号梯上行延时".Q THEN "OUT"."2号梯上行接触器" := TRUE; END_IF;
   IF #_w2 THEN "2号梯数据块"."2号梯初始化楼层中间值byte" := 0; END_IF;
   #_w3 := #_w1 AND "OUT"."2号梯上行接触器";
   #_w4 := #_w3 AND "IN"."2号梯上平层信号" AND NOT "2号梯数据块"."2号梯初始化楼层中间值bool下";   // rising edge of "IN"."2号梯上平层信号"
   "2号梯数据块"."2号梯初始化楼层中间值bool下" := "IN"."2号梯上平层信号";
   IF #_w4 THEN "2号梯数据块"."2号梯初始化楼层中间值byte" := 1 + "2号梯数据块"."2号梯初始化楼层中间值byte"; END_IF;
   IF #_w3 AND ("2号梯数据块"."2号梯初始化楼层中间值byte" = "2号梯数据块"."2号梯初始化楼层") AND "IN"."2号梯下平层信号" THEN
       "OUT"."2号梯上行接触器" := FALSE;
       "OUT"."2号梯低速接触器" := FALSE;
       "OUT"."2号梯电机启动信号" := FALSE;
       "2号梯数据块"."2号梯准备就绪信号" := TRUE;
   END_IF;
END_REGION

REGION Network 4: 2号梯向上初始化
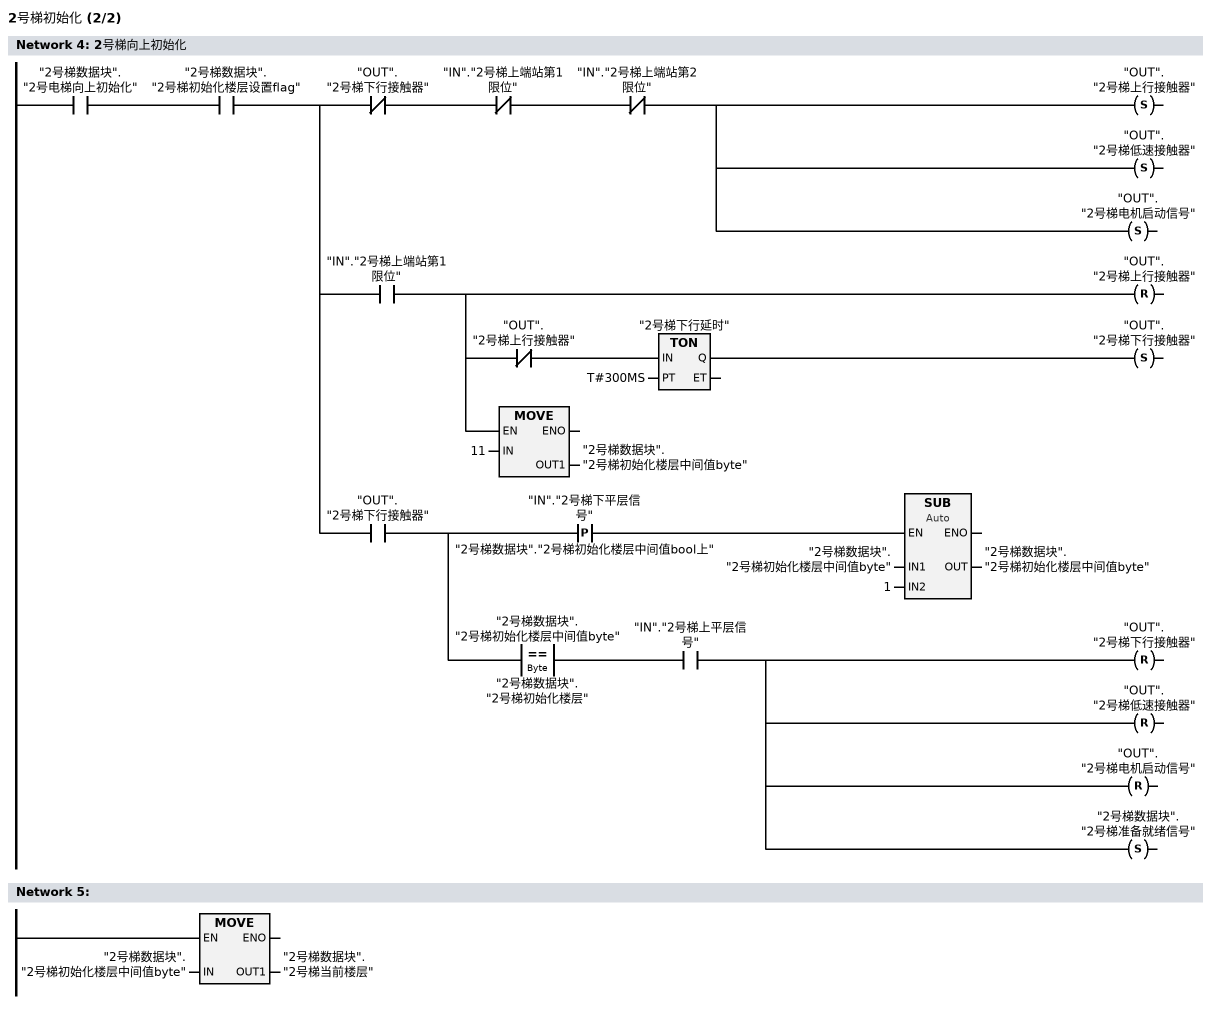
   #_w1 := "2号梯数据块"."2号电梯向上初始化" AND "2号梯数据块"."2号梯初始化楼层设置flag";
   IF #_w1 AND NOT "OUT"."2号梯下行接触器" AND NOT "IN"."2号梯上端站第1限位" AND NOT "IN"."2号梯上端站第2限位" THEN
       "OUT"."2号梯上行接触器" := TRUE;
       "OUT"."2号梯低速接触器" := TRUE;
       "OUT"."2号梯电机启动信号" := TRUE;
   END_IF;
   #_w2 := #_w1 AND "IN"."2号梯上端站第1限位";
   IF #_w2 THEN "OUT"."2号梯上行接触器" := FALSE; END_IF;
   "2号梯下行延时".TON(IN := #_w2 AND NOT "OUT"."2号梯上行接触器", PT := T#300MS);
   IF "2号梯下行延时".Q THEN "OUT"."2号梯下行接触器" := TRUE; END_IF;
   IF #_w2 THEN "2号梯数据块"."2号梯初始化楼层中间值byte" := 11; END_IF;
   #_w3 := #_w1 AND "OUT"."2号梯下行接触器";
   #_w4 := #_w3 AND "IN"."2号梯下平层信号" AND NOT "2号梯数据块"."2号梯初始化楼层中间值bool上";   // rising edge of "IN"."2号梯下平层信号"
   "2号梯数据块"."2号梯初始化楼层中间值bool上" := "IN"."2号梯下平层信号";
   IF #_w4 THEN "2号梯数据块"."2号梯初始化楼层中间值byte" := "2号梯数据块"."2号梯初始化楼层中间值byte" - 1; END_IF;
   IF #_w3 AND ("2号梯数据块"."2号梯初始化楼层中间值byte" = "2号梯数据块"."2号梯初始化楼层") AND "IN"."2号梯上平层信号" THEN
       "OUT"."2号梯下行接触器" := FALSE;
       "OUT"."2号梯低速接触器" := FALSE;
       "OUT"."2号梯电机启动信号" := FALSE;
       "2号梯数据块"."2号梯准备就绪信号" := TRUE;
   END_IF;
END_REGION

REGION Network 5
   RUNG wire#powerrail
      Move(in := "2号梯数据块"."2号梯初始化楼层中间值byte", out1 => "2号梯数据块"."2号梯当前楼层")
   END_RUNG
   // the same network as SCL:
   "2号梯数据块"."2号梯当前楼层" := "2号梯数据块"."2号梯初始化楼层中间值byte";
END_REGION
END_FUNCTION

FUNCTION "2号梯主函数" : Void   // FC9, LAD
{ S7_Optimized_Access := 'TRUE' }
VERSION : 0.1
BEGIN

REGION Network 1
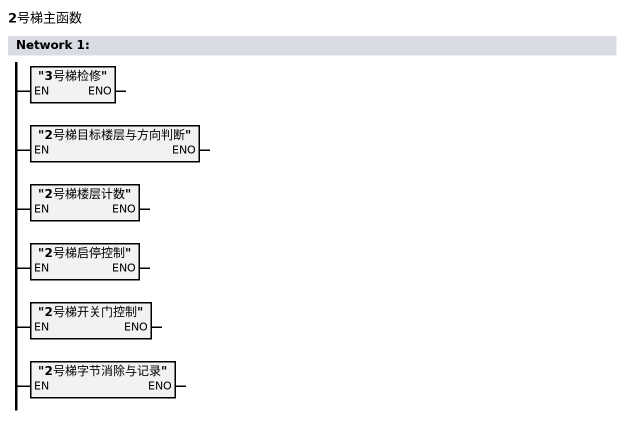
   RUNG wire#powerrail
      "3号梯检修"()
   END_RUNG
   RUNG wire#powerrail
      "2号梯目标楼层与方向判断"()
   END_RUNG
   RUNG wire#powerrail
      "2号梯楼层计数"()
   END_RUNG
   RUNG wire#powerrail
      "2号梯启停控制"()
   END_RUNG
   RUNG wire#powerrail
      "2号梯开关门控制"()
   END_RUNG
   RUNG wire#powerrail
      "2号梯字节消除与记录"()
   END_RUNG
   // the same network as SCL:
   "3号梯检修"();
   "2号梯目标楼层与方向判断"();
   "2号梯楼层计数"();
   "2号梯启停控制"();
   "2号梯开关门控制"();
   "2号梯字节消除与记录"();
END_REGION
END_FUNCTION

FUNCTION "2号梯运行监控模块" : Void   // FC15, LAD
{ S7_Optimized_Access := 'TRUE' }
VERSION : 0.1
BEGIN

REGION Network 1: 2号梯获取当前楼层设置标志位
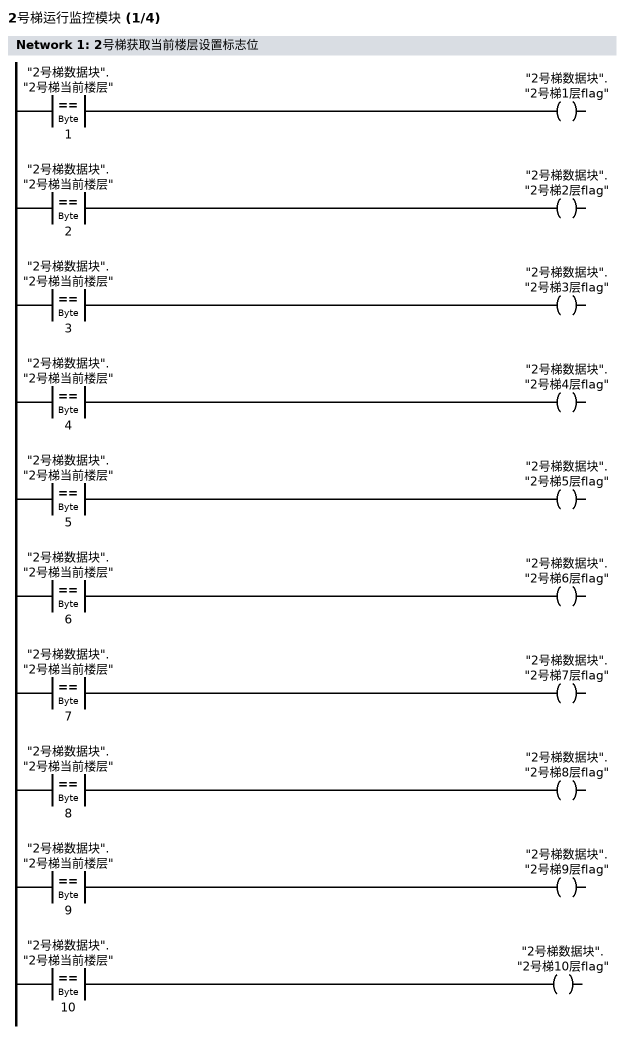
   RUNG wire#powerrail
      { S7_Templates := "SrcType := Byte" } EQ_Contact(in1 := "2号梯数据块"."2号梯当前楼层", in2 := 1)
      Coil( "2号梯数据块"."2号梯1层flag" )
   END_RUNG
   RUNG wire#powerrail
      { S7_Templates := "SrcType := Byte" } EQ_Contact(in1 := "2号梯数据块"."2号梯当前楼层", in2 := 2)
      Coil( "2号梯数据块"."2号梯2层flag" )
   END_RUNG
   RUNG wire#powerrail
      { S7_Templates := "SrcType := Byte" } EQ_Contact(in1 := "2号梯数据块"."2号梯当前楼层", in2 := 3)
      Coil( "2号梯数据块"."2号梯3层flag" )
   END_RUNG
   RUNG wire#powerrail
      { S7_Templates := "SrcType := Byte" } EQ_Contact(in1 := "2号梯数据块"."2号梯当前楼层", in2 := 4)
      Coil( "2号梯数据块"."2号梯4层flag" )
   END_RUNG
   RUNG wire#powerrail
      { S7_Templates := "SrcType := Byte" } EQ_Contact(in1 := "2号梯数据块"."2号梯当前楼层", in2 := 5)
      Coil( "2号梯数据块"."2号梯5层flag" )
   END_RUNG
   RUNG wire#powerrail
      { S7_Templates := "SrcType := Byte" } EQ_Contact(in1 := "2号梯数据块"."2号梯当前楼层", in2 := 6)
      Coil( "2号梯数据块"."2号梯6层flag" )
   END_RUNG
   RUNG wire#powerrail
      { S7_Templates := "SrcType := Byte" } EQ_Contact(in1 := "2号梯数据块"."2号梯当前楼层", in2 := 7)
      Coil( "2号梯数据块"."2号梯7层flag" )
   END_RUNG
   RUNG wire#powerrail
      { S7_Templates := "SrcType := Byte" } EQ_Contact(in1 := "2号梯数据块"."2号梯当前楼层", in2 := 8)
      Coil( "2号梯数据块"."2号梯8层flag" )
   END_RUNG
   RUNG wire#powerrail
      { S7_Templates := "SrcType := Byte" } EQ_Contact(in1 := "2号梯数据块"."2号梯当前楼层", in2 := 9)
      Coil( "2号梯数据块"."2号梯9层flag" )
   END_RUNG
   RUNG wire#powerrail
      { S7_Templates := "SrcType := Byte" } EQ_Contact(in1 := "2号梯数据块"."2号梯当前楼层", in2 := 10)
      Coil( "2号梯数据块"."2号梯10层flag" )
   END_RUNG
   // the same network as SCL:
   "2号梯数据块"."2号梯1层flag" := "2号梯数据块"."2号梯当前楼层" = 1;
   "2号梯数据块"."2号梯2层flag" := "2号梯数据块"."2号梯当前楼层" = 2;
   "2号梯数据块"."2号梯3层flag" := "2号梯数据块"."2号梯当前楼层" = 3;
   "2号梯数据块"."2号梯4层flag" := "2号梯数据块"."2号梯当前楼层" = 4;
   "2号梯数据块"."2号梯5层flag" := "2号梯数据块"."2号梯当前楼层" = 5;
   "2号梯数据块"."2号梯6层flag" := "2号梯数据块"."2号梯当前楼层" = 6;
   "2号梯数据块"."2号梯7层flag" := "2号梯数据块"."2号梯当前楼层" = 7;
   "2号梯数据块"."2号梯8层flag" := "2号梯数据块"."2号梯当前楼层" = 8;
   "2号梯数据块"."2号梯9层flag" := "2号梯数据块"."2号梯当前楼层" = 9;
   "2号梯数据块"."2号梯10层flag" := "2号梯数据块"."2号梯当前楼层" = 10;
END_REGION

REGION Network 2: 2号梯楼层led_a显示
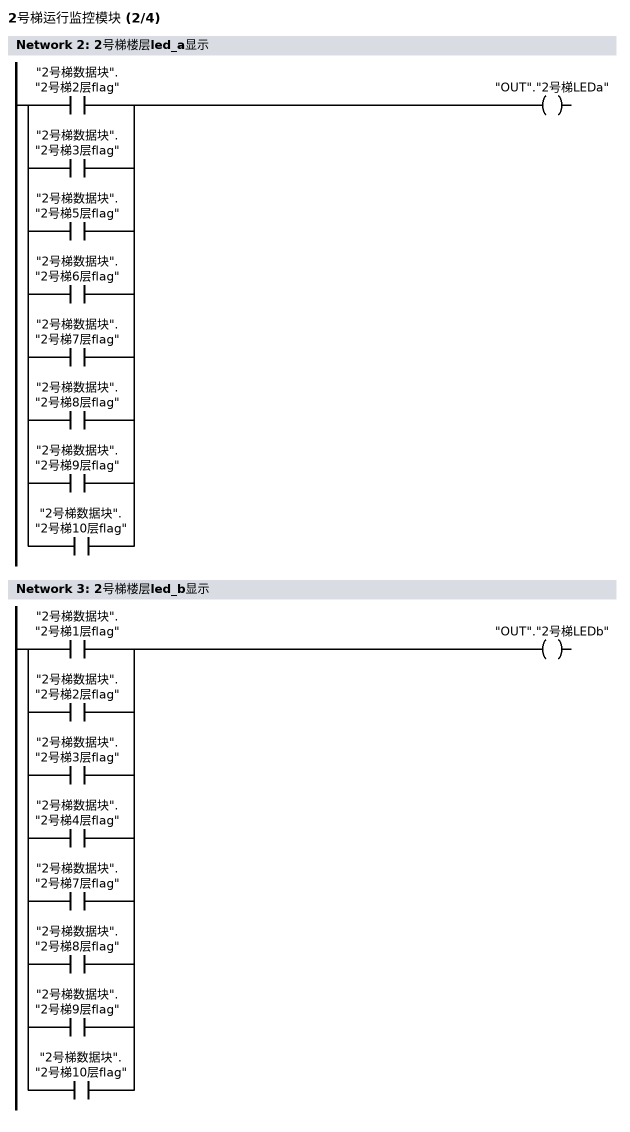
   RUNG wire#powerrail
      Contact( "2号梯数据块"."2号梯2层flag" )
      wire#w1
      Coil( "OUT"."2号梯LEDa" )
   END_RUNG
   RUNG wire#powerrail
      Contact( "2号梯数据块"."2号梯3层flag" )
   END_RUNG wire#w1
   RUNG wire#powerrail
      Contact( "2号梯数据块"."2号梯5层flag" )
   END_RUNG wire#w1
   RUNG wire#powerrail
      Contact( "2号梯数据块"."2号梯6层flag" )
   END_RUNG wire#w1
   RUNG wire#powerrail
      Contact( "2号梯数据块"."2号梯7层flag" )
   END_RUNG wire#w1
   RUNG wire#powerrail
      Contact( "2号梯数据块"."2号梯8层flag" )
   END_RUNG wire#w1
   RUNG wire#powerrail
      Contact( "2号梯数据块"."2号梯9层flag" )
   END_RUNG wire#w1
   RUNG wire#powerrail
      Contact( "2号梯数据块"."2号梯10层flag" )
   END_RUNG wire#w1
   // the same network as SCL:
   "OUT"."2号梯LEDa" := "2号梯数据块"."2号梯2层flag" OR "2号梯数据块"."2号梯3层flag" OR "2号梯数据块"."2号梯5层flag" OR "2号梯数据块"."2号梯6层flag" OR "2号梯数据块"."2号梯7层flag" OR "2号梯数据块"."2号梯8层flag" OR "2号梯数据块"."2号梯9层flag" OR "2号梯数据块"."2号梯10层flag";
END_REGION

REGION Network 3: 2号梯楼层led_b显示
   RUNG wire#powerrail
      Contact( "2号梯数据块"."2号梯1层flag" )
      wire#w1
      Coil( "OUT"."2号梯LEDb" )
   END_RUNG
   RUNG wire#powerrail
      Contact( "2号梯数据块"."2号梯2层flag" )
   END_RUNG wire#w1
   RUNG wire#powerrail
      Contact( "2号梯数据块"."2号梯3层flag" )
   END_RUNG wire#w1
   RUNG wire#powerrail
      Contact( "2号梯数据块"."2号梯4层flag" )
   END_RUNG wire#w1
   RUNG wire#powerrail
      Contact( "2号梯数据块"."2号梯7层flag" )
   END_RUNG wire#w1
   RUNG wire#powerrail
      Contact( "2号梯数据块"."2号梯8层flag" )
   END_RUNG wire#w1
   RUNG wire#powerrail
      Contact( "2号梯数据块"."2号梯9层flag" )
   END_RUNG wire#w1
   RUNG wire#powerrail
      Contact( "2号梯数据块"."2号梯10层flag" )
   END_RUNG wire#w1
   // the same network as SCL:
   "OUT"."2号梯LEDb" := "2号梯数据块"."2号梯1层flag" OR "2号梯数据块"."2号梯2层flag" OR "2号梯数据块"."2号梯3层flag" OR "2号梯数据块"."2号梯4层flag" OR "2号梯数据块"."2号梯7层flag" OR "2号梯数据块"."2号梯8层flag" OR "2号梯数据块"."2号梯9层flag" OR "2号梯数据块"."2号梯10层flag";
END_REGION

REGION Network 4: 2号梯楼层led_c显示
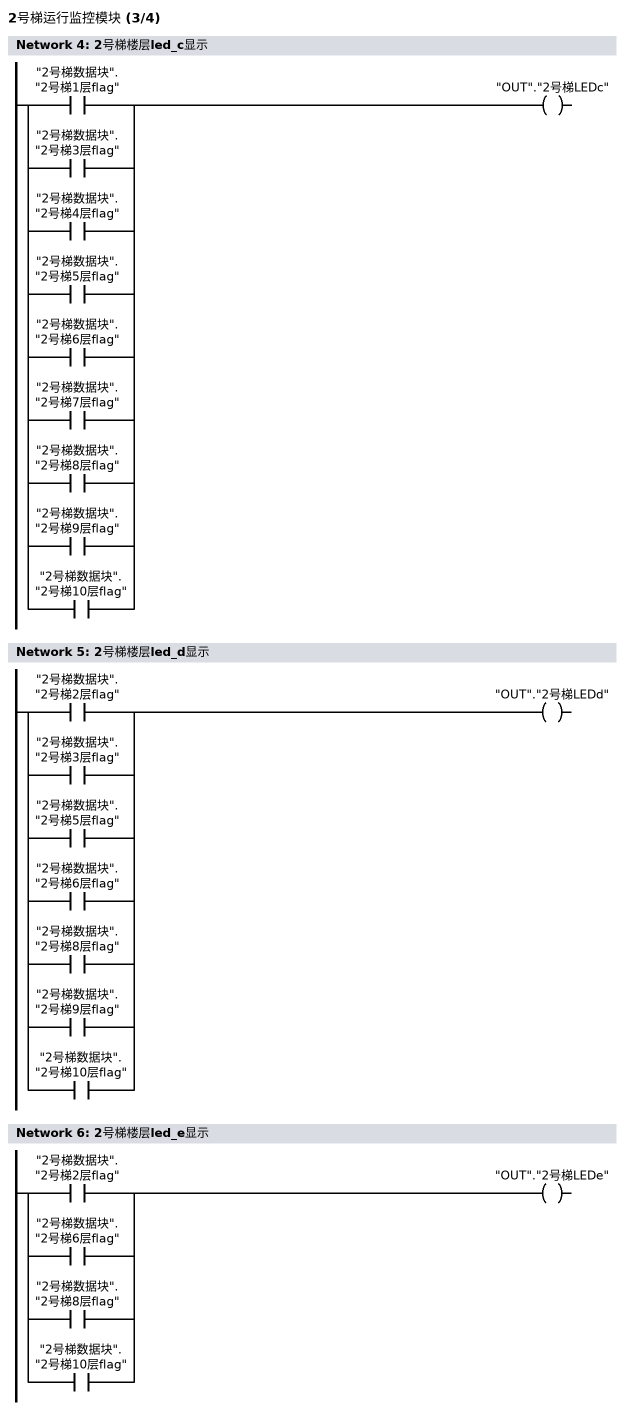
   RUNG wire#powerrail
      Contact( "2号梯数据块"."2号梯1层flag" )
      wire#w1
      Coil( "OUT"."2号梯LEDc" )
   END_RUNG
   RUNG wire#powerrail
      Contact( "2号梯数据块"."2号梯3层flag" )
   END_RUNG wire#w1
   RUNG wire#powerrail
      Contact( "2号梯数据块"."2号梯4层flag" )
   END_RUNG wire#w1
   RUNG wire#powerrail
      Contact( "2号梯数据块"."2号梯5层flag" )
   END_RUNG wire#w1
   RUNG wire#powerrail
      Contact( "2号梯数据块"."2号梯6层flag" )
   END_RUNG wire#w1
   RUNG wire#powerrail
      Contact( "2号梯数据块"."2号梯7层flag" )
   END_RUNG wire#w1
   RUNG wire#powerrail
      Contact( "2号梯数据块"."2号梯8层flag" )
   END_RUNG wire#w1
   RUNG wire#powerrail
      Contact( "2号梯数据块"."2号梯9层flag" )
   END_RUNG wire#w1
   RUNG wire#powerrail
      Contact( "2号梯数据块"."2号梯10层flag" )
   END_RUNG wire#w1
   // the same network as SCL:
   "OUT"."2号梯LEDc" := "2号梯数据块"."2号梯1层flag" OR "2号梯数据块"."2号梯3层flag" OR "2号梯数据块"."2号梯4层flag" OR "2号梯数据块"."2号梯5层flag" OR "2号梯数据块"."2号梯6层flag" OR "2号梯数据块"."2号梯7层flag" OR "2号梯数据块"."2号梯8层flag" OR "2号梯数据块"."2号梯9层flag" OR "2号梯数据块"."2号梯10层flag";
END_REGION

REGION Network 5: 2号梯楼层led_d显示
   RUNG wire#powerrail
      Contact( "2号梯数据块"."2号梯2层flag" )
      wire#w1
      Coil( "OUT"."2号梯LEDd" )
   END_RUNG
   RUNG wire#powerrail
      Contact( "2号梯数据块"."2号梯3层flag" )
   END_RUNG wire#w1
   RUNG wire#powerrail
      Contact( "2号梯数据块"."2号梯5层flag" )
   END_RUNG wire#w1
   RUNG wire#powerrail
      Contact( "2号梯数据块"."2号梯6层flag" )
   END_RUNG wire#w1
   RUNG wire#powerrail
      Contact( "2号梯数据块"."2号梯8层flag" )
   END_RUNG wire#w1
   RUNG wire#powerrail
      Contact( "2号梯数据块"."2号梯9层flag" )
   END_RUNG wire#w1
   RUNG wire#powerrail
      Contact( "2号梯数据块"."2号梯10层flag" )
   END_RUNG wire#w1
   // the same network as SCL:
   "OUT"."2号梯LEDd" := "2号梯数据块"."2号梯2层flag" OR "2号梯数据块"."2号梯3层flag" OR "2号梯数据块"."2号梯5层flag" OR "2号梯数据块"."2号梯6层flag" OR "2号梯数据块"."2号梯8层flag" OR "2号梯数据块"."2号梯9层flag" OR "2号梯数据块"."2号梯10层flag";
END_REGION

REGION Network 6: 2号梯楼层led_e显示
   RUNG wire#powerrail
      Contact( "2号梯数据块"."2号梯2层flag" )
      wire#w1
      Coil( "OUT"."2号梯LEDe" )
   END_RUNG
   RUNG wire#powerrail
      Contact( "2号梯数据块"."2号梯6层flag" )
   END_RUNG wire#w1
   RUNG wire#powerrail
      Contact( "2号梯数据块"."2号梯8层flag" )
   END_RUNG wire#w1
   RUNG wire#powerrail
      Contact( "2号梯数据块"."2号梯10层flag" )
   END_RUNG wire#w1
   // the same network as SCL:
   "OUT"."2号梯LEDe" := "2号梯数据块"."2号梯2层flag" OR "2号梯数据块"."2号梯6层flag" OR "2号梯数据块"."2号梯8层flag" OR "2号梯数据块"."2号梯10层flag";
END_REGION

REGION Network 7: 2号梯楼层led_f显示
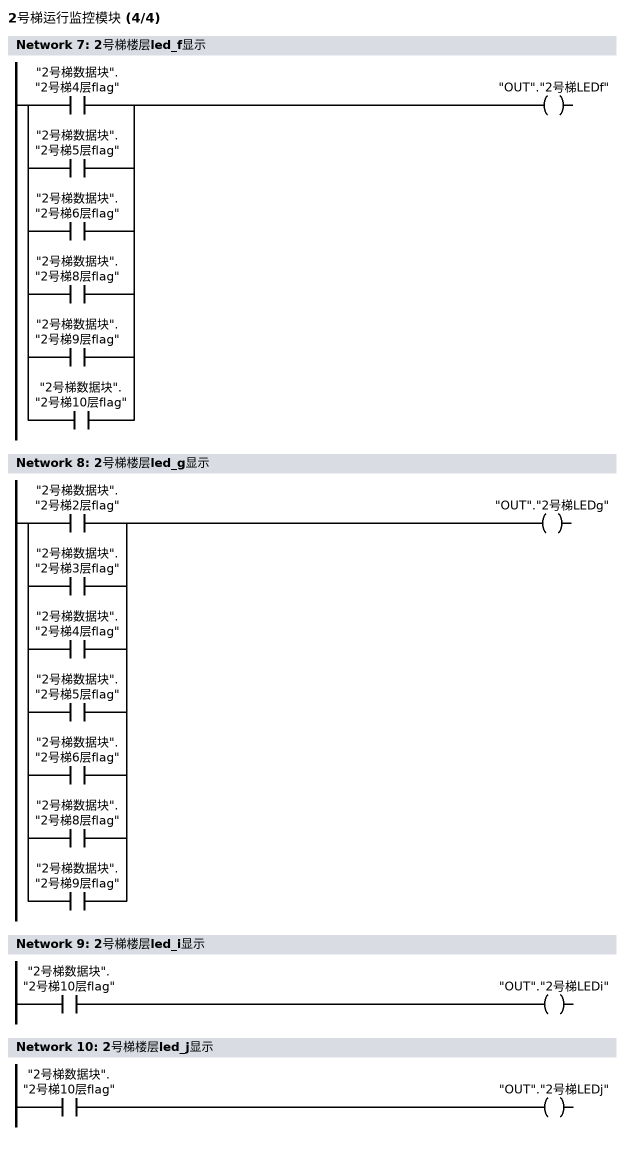
   RUNG wire#powerrail
      Contact( "2号梯数据块"."2号梯4层flag" )
      wire#w1
      Coil( "OUT"."2号梯LEDf" )
   END_RUNG
   RUNG wire#powerrail
      Contact( "2号梯数据块"."2号梯5层flag" )
   END_RUNG wire#w1
   RUNG wire#powerrail
      Contact( "2号梯数据块"."2号梯6层flag" )
   END_RUNG wire#w1
   RUNG wire#powerrail
      Contact( "2号梯数据块"."2号梯8层flag" )
   END_RUNG wire#w1
   RUNG wire#powerrail
      Contact( "2号梯数据块"."2号梯9层flag" )
   END_RUNG wire#w1
   RUNG wire#powerrail
      Contact( "2号梯数据块"."2号梯10层flag" )
   END_RUNG wire#w1
   // the same network as SCL:
   "OUT"."2号梯LEDf" := "2号梯数据块"."2号梯4层flag" OR "2号梯数据块"."2号梯5层flag" OR "2号梯数据块"."2号梯6层flag" OR "2号梯数据块"."2号梯8层flag" OR "2号梯数据块"."2号梯9层flag" OR "2号梯数据块"."2号梯10层flag";
END_REGION

REGION Network 8: 2号梯楼层led_g显示
   RUNG wire#powerrail
      Contact( "2号梯数据块"."2号梯2层flag" )
      wire#w1
      Coil( "OUT"."2号梯LEDg" )
   END_RUNG
   RUNG wire#powerrail
      Contact( "2号梯数据块"."2号梯3层flag" )
   END_RUNG wire#w1
   RUNG wire#powerrail
      Contact( "2号梯数据块"."2号梯4层flag" )
   END_RUNG wire#w1
   RUNG wire#powerrail
      Contact( "2号梯数据块"."2号梯5层flag" )
   END_RUNG wire#w1
   RUNG wire#powerrail
      Contact( "2号梯数据块"."2号梯6层flag" )
   END_RUNG wire#w1
   RUNG wire#powerrail
      Contact( "2号梯数据块"."2号梯8层flag" )
   END_RUNG wire#w1
   RUNG wire#powerrail
      Contact( "2号梯数据块"."2号梯9层flag" )
   END_RUNG wire#w1
   // the same network as SCL:
   "OUT"."2号梯LEDg" := "2号梯数据块"."2号梯2层flag" OR "2号梯数据块"."2号梯3层flag" OR "2号梯数据块"."2号梯4层flag" OR "2号梯数据块"."2号梯5层flag" OR "2号梯数据块"."2号梯6层flag" OR "2号梯数据块"."2号梯8层flag" OR "2号梯数据块"."2号梯9层flag";
END_REGION

REGION Network 9: 2号梯楼层led_i显示
   RUNG wire#powerrail
      Contact( "2号梯数据块"."2号梯10层flag" )
      Coil( "OUT"."2号梯LEDi" )
   END_RUNG
   // the same network as SCL:
   "OUT"."2号梯LEDi" := "2号梯数据块"."2号梯10层flag";
END_REGION

REGION Network 10: 2号梯楼层led_j显示
   RUNG wire#powerrail
      Contact( "2号梯数据块"."2号梯10层flag" )
      Coil( "OUT"."2号梯LEDj" )
   END_RUNG
   // the same network as SCL:
   "OUT"."2号梯LEDj" := "2号梯数据块"."2号梯10层flag";
END_REGION
END_FUNCTION

FUNCTION "2号梯超重与内选" : Void   // FC21, LAD
{ S7_Optimized_Access := 'TRUE' }
VERSION : 0.1
BEGIN

REGION Network 1: 2号梯体重转换
